	16#F85A: F_AX5xErrMsg:= 'F85A =  One cable feedback: Parameter data access error - Timeout';
	16#F85B: F_AX5xErrMsg:= 'F85B =  One cable feedback: Parameter data access error';
	16#F85C: F_AX5xErrMsg:= 'F85C =  One cable feedback: Internal error';
	16#F85D: F_AX5xErrMsg:= 'F85D =  One cable feedback: Encoder status signals an error';
	16#F85E: F_AX5xErrMsg:= 'F85E =  OCT / HpfDSL: Long message bad answer';
	16#F85F: F_AX5xErrMsg:= 'F85F =  OCT / HpfDSL: Shutdown of the encoder failed';
	16#F860: F_AX5xErrMsg:= 'F860 =  OCT / HpfDSL: File write failed.';
	16#F861: F_AX5xErrMsg:= 'F861 =  OCT / HpfDSL: Invalid serial number.';
	16#F862: F_AX5xErrMsg:= 'F862 =  OCT / HpfDSL: No access to the motor temperature sensor.';
	16#F863: F_AX5xErrMsg:= 'F863 =  OCT / HpfDSL: Invalid edge register value.';
	16#F864: F_AX5xErrMsg:= 'F864 =  OCT / HpfDSL: Read cyclic data, Request error';
	16#F865: F_AX5xErrMsg:= 'F865 =  OCT / HpfDSL: Feedback not found.';
	16#F866: F_AX5xErrMsg:= 'F866 =  OCT / HpfDSL: No electronic data sheet found.';
	16#F867: F_AX5xErrMsg:= 'F867 =  OCT / HpfDSL: The electronic data sheet is invalid.';
	16#F868: F_AX5xErrMsg:= 'F868 =  OCT / HpfDSL: User data file invalid.';
	16#F869: F_AX5xErrMsg:= 'F869 =  OCT / HpfDSL: Position offset file invalid.';
	16#F86A: F_AX5xErrMsg:= 'F86A =  OCT / HpfDSL: Commutation offset file invalid.';
	16#F86B: F_AX5xErrMsg:= 'F86B =  OCT / HpfDSL: Invalid file header.';
	16#F86C: F_AX5xErrMsg:= 'F86C =  OCT / HpfDSL: Invalid file.';
	16#F86D: F_AX5xErrMsg:= 'F86D =  OCT / HpfDSL: Position deviation monitoring: Value too many cycles not zero.';
	16#F86E: F_AX5xErrMsg:= 'F86E =  OCT / HpfDSL: Detailed error info';
	16#F86F: F_AX5xErrMsg:= 'F86F =  OCT / HpfDSL: Initial encoder status error';
	16#F870: F_AX5xErrMsg:= 'F870 =  Feedback "AX572x": Encoder not ready';
	16#F872: F_AX5xErrMsg:= 'F872 =  Feedback "AX572x": Position is invalid';
	16#F873: F_AX5xErrMsg:= 'F873 =  Feedback "AX572x": Position is invalid';
	16#F874: F_AX5xErrMsg:= 'F874 =  Feedback "AX572x": Feedbackregister invalid';
	16#F875: F_AX5xErrMsg:= 'F875 =  Feedback "AX572x": Unexpected encoder';
	16#F876: F_AX5xErrMsg:= 'F876 =  Feedback "EnDat 2.2": UART-error';
	16#F877: F_AX5xErrMsg:= 'F877 =  Feedback "AX572x": Out of memory';
	16#F879: F_AX5xErrMsg:= 'F879 =  Feedback "AX572x": Supply voltage';
	16#F87A: F_AX5xErrMsg:= 'F87A =  Feedback "AX572x": Defective Powerup Phase of the feedback system';
	16#F87C: F_AX5xErrMsg:= 'F87C =  Feedback "AX572x": FB protocol not supported';
	16#F87D: F_AX5xErrMsg:= 'F87D =  Feedback "AX572x": Parameter error';
	16#F880: F_AX5xErrMsg:= 'F880 =  HTL: Encoder not ready.';
	16#F881: F_AX5xErrMsg:= 'F881 =  HTL: Error flag active.';
	16#F882: F_AX5xErrMsg:= 'F882 =  HTL: Wrong interface.';
	16#F883: F_AX5xErrMsg:= 'F883 =  HTL: Timeout.';
	16#F8A0: F_AX5xErrMsg:= 'F8A0 =  OCT / HpfDSL: Default state entered.';
	16#F8A1: F_AX5xErrMsg:= 'F8A1 =  OCT / HpfDSL: sHub not supported.';
	16#FA00: F_AX5xErrMsg:= 'FA00 =  Feedback process channel error.';
	16#FA01: F_AX5xErrMsg:= 'FA01 =  Feedback process data channel init error';
	16#FA02: F_AX5xErrMsg:= 'FA02 =  Feedback process channel init command timeout.';
	16#FA03: F_AX5xErrMsg:= 'FA03 =  Feedback process channel init command not idle.';
	16#FA04: F_AX5xErrMsg:= 'FA04 =  Feedback process channel init error.';
	16#FA05: F_AX5xErrMsg:= 'FA05 =  Feedback process channel init error.';
	16#FA06: F_AX5xErrMsg:= 'FA06 =  Feedback process channel init error.';
	16#FA07: F_AX5xErrMsg:= 'FA07 =  Feedback process channel,  unknown feedback type.';
	16#FA40: F_AX5xErrMsg:= 'FA40 =  Feedback process channel error (1Vss)';
	16#FA41: F_AX5xErrMsg:= 'FA41 =  Feedback process channel error (1Vss)';
	16#FA42: F_AX5xErrMsg:= 'FA42 =  Feedback process channel error (1Vss)';
	16#FA43: F_AX5xErrMsg:= 'FA43 =  Feedback process channel error (1Vss)';
	16#FA44: F_AX5xErrMsg:= 'FA44 =  Feedback process channel error (1Vss)';
	16#FA45: F_AX5xErrMsg:= 'FA45 =  Feedback process channel error (1Vss)';
	16#FA46: F_AX5xErrMsg:= 'FA46 =  Feedback process channel error (1Vss)';
	16#FA47: F_AX5xErrMsg:= 'FA47 =  Feedback process channel error (1Vss)';
	16#FA48: F_AX5xErrMsg:= 'FA48 =  Feedback process channel error (1Vss)';
	16#FA49: F_AX5xErrMsg:= 'FA49 =  Feedback process channel error (1Vss)';
	16#FA4A: F_AX5xErrMsg:= 'FA4A =  Feedback process channel error (1Vss)';
	16#FA4B: F_AX5xErrMsg:= 'FA4B =  Feedback process channel error (1Vss)';
	16#FA4C: F_AX5xErrMsg:= 'FA4C =  Feedback process channel error. Failed to set the reference voltage.';
	16#FA4D: F_AX5xErrMsg:= 'FA4D =  Feedback process channel error. Firmware index not valid.';
	16#FA60: F_AX5xErrMsg:= 'FA60 =  Feedback error TTL: System error';
	16#FA61: F_AX5xErrMsg:= 'FA61 =  Feedback error TTL: Unknown state';
	16#FA62: F_AX5xErrMsg:= 'FA62 =  Feedback error TTL: Qudarature encoder error';
	16#FA63: F_AX5xErrMsg:= 'FA63 =  Feedback error TTL: Quadrant init error';
	16#FA64: F_AX5xErrMsg:= 'FA64 =  Feedback error TTL: Reference voltage error';
	16#FA65: F_AX5xErrMsg:= 'FA65 =  Feedback error TTL: Firmware index not supported';
	16#FA80: F_AX5xErrMsg:= 'FA80 =  Feedback "Resolver": Got no timer';
	16#FA81: F_AX5xErrMsg:= 'FA81 =  Feedback "Resolver": Unknown state';
	16#FA82: F_AX5xErrMsg:= 'FA82 =  Feedback "Resolver": Initialisation of the sampling instance failed';
	16#FA83: F_AX5xErrMsg:= 'FA83 =  Feedback "Resolver": Calibration incorrect';
	16#FA84: F_AX5xErrMsg:= 'FA84 =  Feedback "Resolver": Number of poles not supported.';
	16#FA85: F_AX5xErrMsg:= 'FA85 =  Feedback "Resolver": Excitation frequence not supported';
	16#FA86: F_AX5xErrMsg:= 'FA86 =  Feedback "Resolver": Transformation ratio not supported.';
	16#FA87: F_AX5xErrMsg:= 'FA87 =  Feedback "Resolver": Connector not supported.';
	16#FA88: F_AX5xErrMsg:= 'FA88 =  Feedback "Resolver": Invalid ADC configuration';
	16#FA89: F_AX5xErrMsg:= 'FA89 =  Feedback "Resolver": ADC time out';
	16#FA8A: F_AX5xErrMsg:= 'FA8A =  Feedback "Resolver": Hardware does not support a resolver';
	16#FA8B: F_AX5xErrMsg:= 'FA8B =  Feedback "Resolver": Amplitude of the resolver output voltage too large';
	16#FA8C: F_AX5xErrMsg:= 'FA8C =  Feedback "Resolver": Amplitude of the resolver output voltage too low';
	16#FA8D: F_AX5xErrMsg:= 'FA8D =  Feedback "Resolver": Hardware does not support a resolver';
	16#FA8E: F_AX5xErrMsg:= 'FA8E =  Feedback "Resolver": Internal error';
	16#FA8F: F_AX5xErrMsg:= 'FA8F =  Feedback "Resolver": Feedback gear not supported.';
	16#FA90: F_AX5xErrMsg:= 'FA90 =  Feedback "Resolver": Amplitude correction limit exceeded.';
	16#FA91: F_AX5xErrMsg:= 'FA91 =  Feedback "Resolver": Use of reserved parameter.';
	16#FA92: F_AX5xErrMsg:= 'FA92 =  Feedback "Resolver": Offset out of range.';
	16#FA93: F_AX5xErrMsg:= 'FA93 =  Feedback "Resolver": Offset balance failed';
	16#FA94: F_AX5xErrMsg:= 'FA94 =  Feedback "Resolver": Invalid cycle time configuration.';
	16#FA95: F_AX5xErrMsg:= 'FA95 =  Feedback "Resolver": Internal Error';
	16#FA96: F_AX5xErrMsg:= 'FA96 =  Feedback "Resolver": Phase Calibration - Amplitude too low';
	16#FA97: F_AX5xErrMsg:= 'FA97 =  Feedback "Resolver": Phase Calibration - Amplitude too high';
	16#FAB0: F_AX5xErrMsg:= 'FAB0 =  Feedback "MES": Unknown state';
	16#FAB1: F_AX5xErrMsg:= 'FAB1 =  Feedback "MES": Connector not supported.';
	16#FAB2: F_AX5xErrMsg:= 'FAB2 =  Feedback "MES": Invalid ADC configuration';
	16#FAB3: F_AX5xErrMsg:= 'FAB3 =  Feedback "MES": ADC time out';
	16#FAB4: F_AX5xErrMsg:= 'FAB4 =  Feedback "MES": Hardware does not support a MES';
	16#FAB5: F_AX5xErrMsg:= 'FAB5 =  Feedback "MES": Output voltage too high';
	16#FAB6: F_AX5xErrMsg:= 'FAB6 =  Feedback "MES": Output voltage too low';
	16#FAB7: F_AX5xErrMsg:= 'FAB7 =  Feedback "MES": Hardware does not support a MES';
	16#FAB8: F_AX5xErrMsg:= 'FAB8 =  Feedback "MES": Internal error';
	16#FAB9: F_AX5xErrMsg:= 'FAB9 =  Feedback "MES": Feedback gear not supported.';
	16#FABA: F_AX5xErrMsg:= 'FABA =  Feedback "MES": Amplitude correction limit exceeded.';
	16#FABB: F_AX5xErrMsg:= 'FABB =  Feedback "MES": Use of reserved parameter.';
	16#FABC: F_AX5xErrMsg:= 'FABC =  Feedback "MES": Invalid cycle time configuration.';
	16#FC00: F_AX5xErrMsg:= 'FC00 =  Fpga error';
	16#FC01: F_AX5xErrMsg:= 'FC01 =  Fpga error';
	16#FC02: F_AX5xErrMsg:= 'FC02 =  Fpga error';
	16#FC03: F_AX5xErrMsg:= 'FC03 =  Control voltage error: undervoltage';
	16#FC04: F_AX5xErrMsg:= 'FC04 =  Driver unit error: undervoltage';
	16#FC05: F_AX5xErrMsg:= 'FC05 =  Dsp watchdog error.';
	16#FC06: F_AX5xErrMsg:= 'FC06 =  Dsp clock error.';
	16#FC07: F_AX5xErrMsg:= 'FC07 =  ESC clock error.';
	16#FC08: F_AX5xErrMsg:= 'FC08 =  Overcurrent error';
	16#FC09: F_AX5xErrMsg:= 'FC09 =  Deadtime error.';
	16#FC0A: F_AX5xErrMsg:= 'FC0A =  Lock error.';
	16#FC0B: F_AX5xErrMsg:= 'FC0B =  Overcurrent error motor,  short curcuit detection (X13 / X23).';
	16#FC0C: F_AX5xErrMsg:= 'FC0C =  Safety card activated';
	16#FC0D: F_AX5xErrMsg:= 'FC0D =  Shorted coils brake triggerd by the FPGA logic.';
	16#FC0E: F_AX5xErrMsg:= 'FC0E =  Torque off triggerd by the FPGA logic.';
	16#FC0F: F_AX5xErrMsg:= 'FC0F =  FPGA logic: Brake chopper error';
	16#FC10: F_AX5xErrMsg:= 'FC10 =  FPGA logic: Motorcurrent sum error.';
	16#FC11: F_AX5xErrMsg:= 'FC11 =  FPGA logic: Powersupply error.';
	16#FC12: F_AX5xErrMsg:= 'FC12 =  FPGA logic: Umains phase error.';
	16#FC13: F_AX5xErrMsg:= 'FC13 =  FPGA logic:DC link overvoltage';
	16#FC30: F_AX5xErrMsg:= 'FC30 =  Internal error (I2C)';
	16#FC31: F_AX5xErrMsg:= 'FC31 =  Internal error (I2C)';
	16#FC32: F_AX5xErrMsg:= 'FC32 =  Internal error (I2C)';
	16#FC33: F_AX5xErrMsg:= 'FC33 =  Internal error (I2C)';
	16#FC34: F_AX5xErrMsg:= 'FC34 =  Internal error (I2C)';
	16#FC35: F_AX5xErrMsg:= 'FC35 =  Internal error (I2C)';
	16#FC36: F_AX5xErrMsg:= 'FC36 =  Internal error (I2C)';
	16#FC37: F_AX5xErrMsg:= 'FC37 =  Internal communication error';
	16#FC38: F_AX5xErrMsg:= 'FC38 =  Error reading error stack.';
	16#FC39: F_AX5xErrMsg:= 'FC39 =  Error reading operation time.';
	16#FC3A: F_AX5xErrMsg:= 'FC3A =  Error reading eeprom.';
	16#FC3B: F_AX5xErrMsg:= 'FC3B =  Error reading error stack.';
	16#FC3C: F_AX5xErrMsg:= 'FC3C =  Error reading error stack.';
	16#FC3D: F_AX5xErrMsg:= 'FC3D =  Error reading operation time.';
	16#FC3E: F_AX5xErrMsg:= 'FC3E =  Error reading factory settings.';
	16#FC3F: F_AX5xErrMsg:= 'FC3F =  Error reading factory settings.';
	16#FC40: F_AX5xErrMsg:= 'FC40 =  Error saving Hw-Id.';
	16#FC41: F_AX5xErrMsg:= 'FC41 =  Error saving Hw-Id.';
	16#FC42: F_AX5xErrMsg:= 'FC42 =  Error saving factory settings.';
	16#FC43: F_AX5xErrMsg:= 'FC43 =  Error saving factory settings.';
	16#FC44: F_AX5xErrMsg:= 'FC44 =  Error clearing operation time.';
	16#FC45: F_AX5xErrMsg:= 'FC45 =  Error clearing error list.';
	16#FC46: F_AX5xErrMsg:= 'FC46 =  Error reading operation time.';
	16#FC47: F_AX5xErrMsg:= 'FC47 =  Error clearing error stack.';
	16#FC70: F_AX5xErrMsg:= 'FC70 =  Init of the keypad failed.';
	16#FC80: F_AX5xErrMsg:= 'FC80 =  Probe unit error.';
	16#FC81: F_AX5xErrMsg:= 'FC81 =  Probe unit error.';
	16#FC82: F_AX5xErrMsg:= 'FC82 =  Probe unit error.';
	16#FC83: F_AX5xErrMsg:= 'FC83 =  Invalid probe unit configuration';
	16#FC84: F_AX5xErrMsg:= 'FC84 =  Probe unit configuration: Activate signal configuration error.';
	16#FCB0: F_AX5xErrMsg:= 'FCB0 =  LCD Display init failed.';
	16#FCB1: F_AX5xErrMsg:= 'FCB1 =  LDC Display error.';
	16#FCB2: F_AX5xErrMsg:= 'FCB2 =  LDC Display error.';
	16#FCB3: F_AX5xErrMsg:= 'FCB3 =  LCD-Display: Initialisierungsfehler';
	16#FCB4: F_AX5xErrMsg:= 'FCB4 =  LCD-Display: Time out';
	16#FCD0: F_AX5xErrMsg:= 'FCD0 =  Positive limit switch error.';
	16#FCD1: F_AX5xErrMsg:= 'FCD1 =  Negative limit switch error.';
	16#FCD2: F_AX5xErrMsg:= 'FCD2 =  Overspeed error.';
	16#FCD3: F_AX5xErrMsg:= 'FCD3 =  Overspeed error.';
	16#FCD4: F_AX5xErrMsg:= 'FCD4 =  AX5000 utilization error.';
	16#FCD5: F_AX5xErrMsg:= 'FCD5 =  Current limitation: U/F error';
	16#FCD6: F_AX5xErrMsg:= 'FCD6 =  Monitoring functions: Shorted coil / DC brake error';
	16#FCD7: F_AX5xErrMsg:= 'FCD7 =  Maximum output frequency limit exceeded.';
	16#FD00: F_AX5xErrMsg:= 'FD00 =  Motor management: Init failed';
	16#FD01: F_AX5xErrMsg:= 'FD01 =  Motor management: Init failed';
	16#FD03: F_AX5xErrMsg:= 'FD03 =  Brake management error.';
	16#FD04: F_AX5xErrMsg:= 'FD04 =  Periphery voltage missing.';
	16#FD05: F_AX5xErrMsg:= 'FD05 =  Motor management error.';
	16#FD06: F_AX5xErrMsg:= 'FD06 =  Motor management error.';
	16#FD07: F_AX5xErrMsg:= 'FD07 =  Motor overtemperature shut down.';
	16#FD08: F_AX5xErrMsg:= 'FD08 =  Motor management: Drive type don"t match.';
	16#FD09: F_AX5xErrMsg:= 'FD09 =  Motor management: Motor type don"t match.';
	16#FD0A: F_AX5xErrMsg:= 'FD0A =  Configured channel peak current is greater than the motor peak current.';
	16#FD0B: F_AX5xErrMsg:= 'FD0B =  Configured channel peak current is greater than the amplifier channel peak current.';
	16#FD0C: F_AX5xErrMsg:= 'FD0C =  Configured channel current is greater than the motor coninuous stall current.';
	16#FD0D: F_AX5xErrMsg:= 'FD0D =  Configured channel current is greater than the amplifier rated current.';
	16#FD0E: F_AX5xErrMsg:= 'FD0E =  Invalid total output current.';
	16#FD0F: F_AX5xErrMsg:= 'FD0F =  Motor brake: Current monitoring error.';
	16#FD10: F_AX5xErrMsg:= 'FD10 =  Periphery voltage too high.';
	16#FD11: F_AX5xErrMsg:= 'FD11 =  Periphery voltage too low.';
	16#FD12: F_AX5xErrMsg:= 'FD12 =  Unknown constraint IDN';
	16#FD13: F_AX5xErrMsg:= 'FD13 =  Too low dielectric strength of the motor winding.';
	16#FD14: F_AX5xErrMsg:= 'FD14 =  Constraint check failed.';
	16#FD15: F_AX5xErrMsg:= 'FD15 =  The maximum feedback frequency is too high.';
	16#FD16: F_AX5xErrMsg:= 'FD16 =  Unknown feedback system.';
	16#FD17: F_AX5xErrMsg:= 'FD17 =  Motor overload shutdown.';
	16#FD18: F_AX5xErrMsg:= 'FD18 =  Motorbrake current: Measuring error';
	16#FD19: F_AX5xErrMsg:= 'FD19 =  A/D-Converter: Peripheral voltage - measuring error';
	16#FD1A: F_AX5xErrMsg:= 'FD1A =  A/D-Converter: Motor temperature - measuring error';
	16#FD1B: F_AX5xErrMsg:= 'FD1B =  Motor cont. stall torque > peak torque';
	16#FD1C: F_AX5xErrMsg:= 'FD1C =  ASM don"t support"s usage of P-0-0077';
	16#FD1D: F_AX5xErrMsg:= 'FD1D =  Invalid torque characteristic data.';
	16#FD1E: F_AX5xErrMsg:= 'FD1E =  Invalid inductance characteristic data.';
	16#FD1F: F_AX5xErrMsg:= 'FD1F =  Got no memory.';
	16#FD20: F_AX5xErrMsg:= 'FD20 =  Motor management: Invalid motor data.';
	16#FD21: F_AX5xErrMsg:= 'FD21 =  Motor management: Voltage error';
	16#FD22: F_AX5xErrMsg:= 'FD22 =  Motor management: Current error';
	16#FD40: F_AX5xErrMsg:= 'FD40 =  Power management: Init failed';
	16#FD41: F_AX5xErrMsg:= 'FD41 =  Mains supply: U mains too high.';
	16#FD42: F_AX5xErrMsg:= 'FD42 =  Mains supply: U mains too low.';
	16#FD43: F_AX5xErrMsg:= 'FD43 =  Mains supply: Power down.';
	16#FD44: F_AX5xErrMsg:= 'FD44 =  Mains supply: Phase error.';
	16#FD45: F_AX5xErrMsg:= 'FD45 =  Continous power internal brake resistor too low.';
	16#FD46: F_AX5xErrMsg:= 'FD46 =  Power management error.';
	16#FD47: F_AX5xErrMsg:= 'FD47 =  Power management error.';
	16#FD48: F_AX5xErrMsg:= 'FD48 =  Power management error.';
	16#FD49: F_AX5xErrMsg:= 'FD49 =  IGBT temperature measuring error.';
	16#FD4A: F_AX5xErrMsg:= 'FD4A =  IGBT temperature measuring error.';
	16#FD4B: F_AX5xErrMsg:= 'FD4B =  DC link undervoltage.';
	16#FD4C: F_AX5xErrMsg:= 'FD4C =  DC link overvoltage';
	16#FD4D: F_AX5xErrMsg:= 'FD4D =  Cooling error shut down.';
	16#FD4E: F_AX5xErrMsg:= 'FD4E =  Control voltage error';
	16#FD4F: F_AX5xErrMsg:= 'FD4F =  Overvoltage error.';
	16#FD50: F_AX5xErrMsg:= 'FD50 =  Undervoltage error.';
	16#FD51: F_AX5xErrMsg:= 'FD51 =  Power supply phase error.';
	16#FD52: F_AX5xErrMsg:= 'FD52 =  Unknown internal brake resistor.';
	16#FD53: F_AX5xErrMsg:= 'FD53 =  U_mains power up after mains power failure.';
	16#FD54: F_AX5xErrMsg:= 'FD54 =  Unknown nominal device current.';
	16#FD55: F_AX5xErrMsg:= 'FD55 =  AX5021: Brake resistor overtemperature shut down';
	16#FD56: F_AX5xErrMsg:= 'FD56 =  Error Power Management: Transfer error, unknown channel.';
	16#FD57: F_AX5xErrMsg:= 'FD57 =  Error Power Management: Load resistor active and axis enabled';
	16#FD58: F_AX5xErrMsg:= 'FD58 =  Error Power Management: Check external dc link connection';
	16#FD59: F_AX5xErrMsg:= 'FD59 =  Error Power Management: Wrong external brake resistor found';
	16#FD5A: F_AX5xErrMsg:= 'FD5A =  Power Management: Overcurrent - dc link connection';
	16#FD80: F_AX5xErrMsg:= 'FD80 =  System time underflow error.';
	16#FD81: F_AX5xErrMsg:= 'FD81 =  Wrong timer pointer.';
	16#FD82: F_AX5xErrMsg:= 'FD82 =  Out of timer.';
	16#FD83: F_AX5xErrMsg:= 'FD83 =  Invalid identity object type.';
	16#FD84: F_AX5xErrMsg:= 'FD84 =  Invalid firmware index.';
	16#FD85: F_AX5xErrMsg:= 'FD85 =  Feedback firmware checksum error.';
	16#FD86: F_AX5xErrMsg:= 'FD86 =  System timer underflow.';
	16#FD87: F_AX5xErrMsg:= 'FD87 =  Error: Out of system timer.';
	16#FD88: F_AX5xErrMsg:= 'FD88 =  Found not supported hardware type.';
	16#FD89: F_AX5xErrMsg:= 'FD89 =  Safety card type not supported.';
	16#FD8A: F_AX5xErrMsg:= 'FD8A =  Option card: Type not supported';
	16#FD8B: F_AX5xErrMsg:= 'FD8B =  Option card: Interface Id is not supported.';
	16#FD8C: F_AX5xErrMsg:= 'FD8C =  Option card: Channel count is not supported.';
	16#FD8D: F_AX5xErrMsg:= 'FD8D =  Invalid identity object';
	16#FD8E: F_AX5xErrMsg:= 'FD8E =  Optioncard: Interface of the FPGA 2 not supported';
	16#FDB0: F_AX5xErrMsg:= 'FDB0 =  Customer specific function: Init failed.';
	16#FDC0: F_AX5xErrMsg:= 'FDC0 =  Internal command state machine error.';
	16#FDC1: F_AX5xErrMsg:= 'FDC1 =  Internal command state machine error.';
	16#FDC2: F_AX5xErrMsg:= 'FDC2 =  Internal command state machine error.';
	16#FDC3: F_AX5xErrMsg:= 'FDC3 =  Internal command state machine error.';
	16#FDD0: F_AX5xErrMsg:= 'FDD0 =  Safety card: Unknown hardware type.';
	16#FDD1: F_AX5xErrMsg:= 'FDD1 =  Safety: internal error, out of memory';
	16#FDD2: F_AX5xErrMsg:= 'FDD2 =  Safety: internal error, got no timer';
	16#FDD3: F_AX5xErrMsg:= 'FDD3 =  Safety switch off while the axis was enabled.';
	16#FDD4: F_AX5xErrMsg:= 'FDD4 =  Configured safety option don"t match';
	16#FDD5: F_AX5xErrMsg:= 'FDD5 =  The basic unit of the drive dont supports a safety option.';
	16#FDD6: F_AX5xErrMsg:= 'FDD6 =  Safety Option: Not supported firmware index.';
	16#FDD7: F_AX5xErrMsg:= 'FDD7 =  Safety slot: No safety or dummy card inserted';
	16#FDD8: F_AX5xErrMsg:= 'FDD8 =  Safety slot: Wrong safety or dummy card inserted';
	16#FDD9: F_AX5xErrMsg:= 'FDD9 =  Safety card: safety card activated - internal reaction';
	16#FDDA: F_AX5xErrMsg:= 'FDDA =  Safety slot: Wrong safety card AX5805 or AX5806 inserted';
	16#FDDB: F_AX5xErrMsg:= 'FDDB =  Safety card: Internal error.';
	16#FFFE: F_AX5xErrMsg:= 'FFFE =  Missing implementation!';
	
ELSE
	F_AX5xErrMsg := UINT_TO_STRING(uiDriveError);
	F_AX5xErrMsg := concat(F_AX5xErrMsg, ' Unknown Error code');
END_CASE
F_AX5xErrMsg := F_AX5xErrMsg;

END_FUNCTION

// ---- POUs/P_ModeStateManager.TcPOU
//==================================================================================================
//							Beckhoff Automation Poland
//									2.11.2018
//	Zarzadzeni trybami pracy i komendami - Satate Machine
// 	v1.2	|| TC v 3.1.4022.25		|| - dodano Initialization 
// 	v1.1	|| TC v 3.1.4022.4		|| - Aktualizacja - dodano test Abort z HMI 
// 	v1.0	|| TC v 3.1.4022.4		|| - Pierwsza wersja
//==================================================================================================
PROGRAM P_ModeStateManager
VAR
	//	GVL_Machine - HMI handling
	bHMIModeRequest_Automatic			: BOOL;
	bHMIModeRequest_Manual				: BOOL;
	bHMIModeRequest_Maintenance			: BOOL;
	
	bHMICommandRequest_Run				: BOOL;
	bHMICommandRequest_Stop				: BOOL;
	bHMICommandRequest_Reset			: BOOL;
	bHMICommandRequest_Restart			: BOOL;
	bHMICommandRequest_Abort			: BOOL;
	// Rising edge detection
	rtButtonAutomatic					: R_TRIG;
	rtButtonManual						: R_TRIG;
	rtButtonMaintenance					: R_TRIG;
	rtButtonStart						: R_TRIG;
	rtButtonReset						: R_TRIG;
	rtButtonStop						: R_TRIG;
	// State change permissions
	bAllowChangeToManual				: BOOL;
	bAllowChangeToMaintenance			: BOOL;
	bAllowChangeToAutomatic				: BOOL;
END_VAR

// Triggers
rtButtonAutomatic(CLK:= bHMIModeRequest_Automatic);
rtButtonManual(CLK:= bHMIModeRequest_Manual);
rtButtonMaintenance(CLK:= bHMIModeRequest_Maintenance);
rtButtonStart(CLK:= GVL_IO.di_PBStart OR bHMICommandRequest_Run);
rtButtonStop(CLK:= GVL_IO.di_PBStop OR bHMICommandRequest_Stop);
rtButtonReset(CLK:= GVL_IO.di_PBReset OR bHMICommandRequest_Reset);

// SAFETY niezaleznie
IF NOT GVL_IO.bSAFETY_PermissionSS1 OR bHMICommandRequest_Abort THEN
	GVL_Machine.eCommand						:= E_MachineCommand.eAbort;
	GVL_Machine.eState							:= E_MachineState.eAborted;
END_IF
		
CASE GVL_Machine.eMode OF 

	E_MachineMode.eInitialization:

		// Reset just in case of init error
		P_Initialization(bReset := (P_Initialization.bError AND rtButtonReset.Q), bTestMode := );
		IF P_Initialization.bInitialized THEN
			// Choose mode to go
			GVL_Machine.eMode						:= E_MachineMode.eManual;
		END_IF
		
	E_MachineMode.eAutomatic:

		// Zmiana trybu tylko gdy maszyna nie jest w Running
		IF GVL_Machine.eState <> E_MachineState.eRunning THEN
			IF rtButtonMaintenance.Q THEN
				GVL_Machine.eState				:= E_MachineState.eIdle;
				GVL_Machine.eMode				:= E_MachineMode.eMaintenance;
			END_IF
		END_IF

		//==============================================
		IF rtButtonStart.Q THEN 
			GVL_Machine.eCommand 	:= E_MachineCommand.eRun;
		END_IF

		IF rtButtonReset.Q AND GVL.bRestartRequired THEN
			GVL_Machine.eCommand	:= E_MachineCommand.eRestart;
		END_IF
		
		IF rtButtonReset.Q AND NOT GVL.bRestartRequired THEN
			GVL_Machine.eCommand	:= E_MachineCommand.eReset;
		END_IF
		
		IF GVL.bGeneralError OR GVL.bGeneralFatalError OR rtButtonStop.Q THEN
			GVL_Machine.eCommand	:= E_MachineCommand.eStop ;
		END_IF
		
	E_MachineMode.eMaintenance, E_MachineMode.eManual:
	
		// Reset, Restart, Error - not used
		
		// Zmiana trybu tylko gdy maszyna nie jest w Running
		IF GVL_Machine.eState <> E_MachineState.eRunning THEN
			IF rtButtonAutomatic.Q (* OR sth *) THEN
				GVL_Machine.eState				:= E_MachineState.eIdle;
				GVL_Machine.eMode				:= E_MachineMode.eAutomatic;
			END_IF
		END_IF
		
		//==============================================
		IF rtButtonStart.Q THEN 
			GVL_Machine.eCommand 	:= E_MachineCommand.eRun;
		END_IF

		IF rtButtonReset.Q AND GVL.bRestartRequired THEN
			GVL_Machine.eCommand	:= E_MachineCommand.eRestart;
		END_IF
		
		IF rtButtonReset.Q AND NOT GVL.bRestartRequired THEN
			GVL_Machine.eCommand	:= E_MachineCommand.eReset;
		END_IF
		
		IF rtButtonStop.Q THEN
			GVL_Machine.eCommand	:= E_MachineCommand.eStop ;
		END_IF

END_CASE

ACTION Act_CollectMachineState:
// Action to decide global machine state
GVL_Machine.eState; // :=
END_ACTION

ACTION Act_ModeChangeSelector:
bAllowChangeToManual 				:= NOT (P_Template.eMachineState <> E_MachineState.eRunning); //
bAllowChangeToMaintenance;
bAllowChangeToAutomatic;
END_ACTION

END_PROGRAM

// ---- POUs/P_Initialization.TcPOU
//==================================================================================================
//							Beckhoff Automation Poland
//									2.11.2018
//	Program inicjalizujacy prace maszyny - powinien byc wykonywany tylko w trybie E_MachineMode.eInitialization
//	Przejscie do innych trybow powinno byc mozliwe po wystawieniu flagi bInitialized
//	Program podczas inicjalizacji tlumi globalne flagi: GVL.bMuteGeneralError i GVL.bMuteGeneralFatalError
//	Reset mozliwy tylko w przypadku bledu.
//	Zawiera opsje testu - ignorujemy wowczas bledy i przechodzimy od razu do stanu bInitialized
// 	v1.0	|| TC v 3.1.4022.25		|| - Pierwsza wersja
//==================================================================================================
PROGRAM P_Initialization
VAR_INPUT
	bReset					: BOOL;
	bTestMode				: BOOL;				// Deactivate error detecton - go to initialized
END_VAR
VAR_OUTPUT
	bInitialized			: BOOL;
	bBusy					: BOOL;
	bError					: BOOL;
END_VAR
VAR
	iStep					: INT;
	rtReset					: R_TRIG;
	rtError					: R_TRIG;
	tonWatchdog				: TON;
END_VAR

// Wait some time to initialize
tonWatchdog(IN:= bBusy, PT:= T#1M, Q=> , ET=> );
rtError(CLK:= tonWatchdog.Q, Q=> );

IF rtError.Q THEN
	iStep							:= 1000;
END_IF

// Reset - reinitialize
rtReset(CLK:= bReset, Q=> );

IF bTestMode THEN
	iStep							:= 500;
END_IF

CASE iStep OF

	0: // Idle
	
		iStep	 					:= iStep + 10;
	
	10: 
	
		IF P_SystemInfo.bOK THEN
			iStep 					:= iStep + 10;
		ELSE
			// There is problem with System - usually persistent data
			P_SystemInfo.bConfirm 	:= bReset;
		END_IF
	
	20:

		IF P_EtherCAT_Diag.bOK THEN
			iStep 					:= iStep + 10;
		END_IF

	30:

		IF P_Checks.bOK THEN
			iStep 					:= iStep + 10;
		END_IF
		
	40:

		IF P_TaskInfo.bOK THEN
			iStep 					:= iStep + 10;
		END_IF
		
	50:
	// Serial No, etc
		iStep 						:= 500;
		
	500: // Initialized
	
		;
	
	1000: // Error step, wait for reset
	
		IF rtReset.Q THEN
			P_SystemInfo.bConfirm 	:= TRUE;
			iStep 					:= 0;
		END_IF;

END_CASE

bBusy 								:= iStep < 500;
bError 								:= iStep = 1000;
bInitialized						:= iStep = 500;

// Mute Errors during init phase
GVL.bMuteGeneralError				:= bBusy;
GVL.bMuteGeneralFatalError			:= bBusy;

END_PROGRAM

// ---- POUs/POUsAxisOnline/AX8000/FB_HoldingBrakeCtrlAX8000.TcPOU
//==================================================================================================
//							Beckhoff Automation Poland
//									12.04.2018
//	Blok funkcyjny kontroli luzownika w silniku podpietym do AX8000. Przewaga ForceLock
//	Dzialania na obiekcie: 3000:07 Motor brake force
//	Index:			AxisMainSlot: 16#3000 (Ch A)/ 16#3400 (Ch B)
//	Subindex:		16#07
//	Datatype:		ENUM (INT16)
//	Enum Value:		0 (0x00): 	Release_force
//					1 (0x01): 	Force_lock
//					2 (0x02): 	Force_unlock
//
//  v1.0	|| TC v 3.1.4022.16		|| - pierwsza wersja
//==================================================================================================
FUNCTION_BLOCK FB_HoldingBrakeCtrlAX8000
VAR_INPUT
	bForceLock 						: BOOL;								// 
	bForceUnlock					: BOOL;								// 
	stDriveRef						: ST_DriveRef;
END_VAR
VAR_OUTPUT
	bBusy							: BOOL;
	bError							: BOOL; 							// General error: parameter or CoE read.
																		// If bError = TRUE and bInitialized = FALSE - error during read motor data.
																		// If bError = TRUE and bInitialized = TRUE and (iAdsErrId <> 0 or iCANopenErrId <> 0) then I2T read error
																		// If bError = TRUE and bInitialized = TRUE and iAdsErrId = 0 and iCANopenErrId = 0 then parameter error: rTorqueLimit outside permitted range rTorqueLimitLow..rTorqueLimitHigh or Empty stDriveRef
	iAdsErrId						: UINT;								// Forwarded output FB_CoERead_ByDriveRef
	iCANopenErrId					: UINT;								// Forwarded output FB_CoERead_ByDriveRef
END_VAR
VAR
	bExecute						: BOOL;
	iMotorBrakeForce				: INT;								// 0 - Release_force, 1 - Force_lock, 2 - Force_unlock
	rtForceLock						: R_TRIG;
	rtForceUnlock					: R_TRIG;
	ftForceLock						: F_TRIG;
	ftForceUnlock					: F_TRIG;
	fbForceLockUnlock				: FB_CoEWrite_ByDriveRef;
END_VAR

{region "Call triggers"}
//======================= Call triggers =========================
rtForceLock(CLK:= bForceLock);
ftForceLock(CLK:= bForceLock);
rtForceUnlock(CLK:= bForceUnlock);
ftForceUnlock(CLK:= bForceUnlock);
bExecute								:= rtForceLock.Q OR ftForceLock.Q OR rtForceUnlock.Q OR ftForceUnlock.Q;
//===============================================================
{endregion}
{region "Main code"}
//========================= Main code ===========================
IF bExecute THEN
	iMotorBrakeForce 						:= 0;										// Clear value
	iMotorBrakeForce.1 						:= bForceUnlock;							// Set force unlock bit
	iMotorBrakeForce 						:= SEL(bForceLock, iMotorBrakeForce, 1);	// Set force lock bit, it has higher priority than unlock
END_IF

fbForceLockUnlock(	stDriveRef				:= stDriveRef, 
					nIndex					:= 16#3000 + (stDriveRef.nDriveNo * 16#400), 
					nSubIndex				:= 16#07, 
					pSrcBuf					:= ADR(iMotorBrakeForce), 
					cbBufLen				:= SIZEOF(iMotorBrakeForce), 
					bExecute				:= bExecute,
					bBusy					=> bBusy, 
					bError					=> bError, 
					iAdsErrId				=> iAdsErrId, 
					iCANopenErrId			=> iCANopenErrId);
//===============================================================
{endregion}

END_FUNCTION_BLOCK

// ---- POUs/POUsAxisOnline/AX8000/FB_McAxisOnlineAX8000.TcPOU
//==================================================================================================
//							Beckhoff Automation Poland
//									7.12.2018
//	Wszystkomajacy blok funkcyjny do sterowania osia, 
//	wymagane biblioteki: Tc2_EtherCAT, Tc2_MC2_Drive, Tc2_MC2
//  v1.5	|| TC v 3.1.4022.27		|| - dodane opisy bledow w formie zmiennych typu string
// 	v1.4 	|| TC v 3.1.4022.20	 	|| - ACT_MotorMonitoring - only for real axis
// 	v1.3 	|| TC v 3.1.4022.16	 	|| - spojne z AX5000
// 	v1.2 	|| TC v 3.1.4022.16	 	|| - Added ACT_SetPositionIO, migration part of logic from ACT_SetPosition to ACT_SetPositionIO
// 	v1.1 	|| TC v 3.1.4022.16	 	|| - ACT_MotorMonitoring - is executing always, ACT_Initialization - optimalization
// 	v1.0 	|| TC v 3.1.4022.16	 	|| - first edition
//==================================================================================================
{attribute 'reflection'}
FUNCTION_BLOCK FB_McAxisOnlineAX8000
VAR_IN_OUT
	stMcAxisOnline						: ST_McAxisOnline;
	Axis								: AXIS_REF;
END_VAR
VAR
	mcPower								: MC_Power;
	mcStop								: MC_Stop;
	mcHalt								: MC_Halt;
	mcStopSS1							: MC_Stop;
	mcStopSS2							: MC_Stop;
	mcReset								: MC_Reset;
	mcHome								: MC_Home;
	mcSetPosition						: MC_SetPosition;
	fbSetPositionOffset					: FB_CoEAX8000SetPositionOffset;
	mcJog								: MC_Jog;

	mcMoveAbsolute						: MC_MoveAbsolute;
	mcMoveRelative						: MC_MoveRelative;
	mcMoveVelocity						: MC_MoveVelocity;
	mcMoveModulo						: MC_MoveModulo;
	mcMoveAbsolute2						: MC_MoveAbsolute;
	mcMoveRelative2						: MC_MoveRelative;
	mcMoveVelocity2						: MC_MoveVelocity;
	mcMoveModulo2						: MC_MoveModulo;

	fbMotorMonitoring					: FB_MotorMonitoringAX8000;
	fbHoldingBrakeCtrl					: FB_HoldingBrakeCtrlAX8000;
	fbNcLimitSwitch						: FB_NcSWLimitSwitchCtrl;
	tonGetDriveDiag						: TON;
	fbReadChannelErrorCode				: FB_ReadChannelErrorCodeAX8000;
	
	mcReadDriveAddress					: MC_ReadDriveAddress;
	mcReadParameterSet					: MC_ReadParameterSet;
	fbGetDriveRef						: FB_GetDriveRef;

	// Internal
	bInitialized						: BOOL;
	bCommError							: BOOL;
	bReadParameterError					: BOOL;
	bInitError							: BOOL;
	bDriveError							: BOOL;
	bFBError							: BOOL;
	
// Initialization
	iInitStep							: INT;
	bInitializationError				: BOOL;
	wInitializationErrorCounter			: WORD;
	bDriveAddressReady					: BOOL;
	bDriveRefReady						: BOOL;
	bReadParameterSetReady				: BOOL;
	tonDelay							: TON;
// Re init
	udiOnlineChangeCntOld				: UDINT;
	bOnlineChangeDetected				: BOOL;
	bReInit								: BOOL;
	bReInitialized						: BOOL;
	bReInitializationError				: BOOL;
	{attribute 'instance-path'}
	{attribute 'noinit'}
	sInstancePath						: STRING;
END_VAR

// Device dependent initialization 
ACT_Initialization();
// Device independent commands, mostly NC 
ACT_States();
ACT_SWLimitSwitch();
ACT_Stop();
ACT_Power();
ACT_Homing();
ACT_Jog();
ACT_Move();
ACT_Reset();
ACT_SetPosition();
// Device dependent commands
// Motor monitoring possible only with real axis
IF NOT Axis.Status.OpMode.SimulationAxis THEN
	ACT_MotorMonitoring();
END_IF
// Device dependent commands, possible only on real axis after complete initialization
IF bInitialized AND NOT Axis.Status.OpMode.SimulationAxis THEN
	ACT_SetPositionIO();
	ACT_DriveDiag();
	ACT_HoldingBrakeCtrl();
END_IF

// Device independent error collection
ACT_ErrorCollection();

ACTION ACT_DriveDiag:
// Auto update when drive error
tonGetDriveDiag(IN:= stMcAxisOnline.stError.bDriveError AND NOT tonGetDriveDiag.Q, PT:= T#5S, Q=> , ET=> );

fbReadChannelErrorCode(	bExecute				:= stMcAxisOnline.stChannelErrorCode.bExecute OR tonGetDriveDiag.Q,
						stDriveRef				:= stMcAxisOnline.stDriveRef,
						bBusy					=> stMcAxisOnline.stChannelErrorCode.bBusy,
						bError					=> stMcAxisOnline.stChannelErrorCode.bError,
						iAdsErrId				=> stMcAxisOnline.stChannelErrorCode.uiAdsErrId,
						iCANopenErrId			=> stMcAxisOnline.stChannelErrorCode.uiSecErrId,
						uiChannelErrorCode		=> stMcAxisOnline.stChannelErrorCode.uiChannelErrorCode,
						uiChannelErrorCodeHex	=> stMcAxisOnline.stChannelErrorCode.uiChannelErrorCodeHex);
END_ACTION

ACTION ACT_ErrorCollection:
// Error flags
stMcAxisOnline.stError.bDriveError					:= Axis.Status.DriveDeviceError;

stMcAxisOnline.stError.bNcError						:= Axis.Status.Error;

stMcAxisOnline.stError.bFBError						:= stMcAxisOnline.mcPower.bError OR stMcAxisOnline.mcReset.bError OR stMcAxisOnline.mcHome.bError OR stMcAxisOnline.mcJog.bError
													OR stMcAxisOnline.mcHalt.bError OR stMcAxisOnline.mcStop.bError OR stMcAxisOnline.mcSS1.bError OR stMcAxisOnline.mcSS2.bError
													OR stMcAxisOnline.mcMoveAbsolute.bError OR stMcAxisOnline.mcMoveRelative.bError OR stMcAxisOnline.mcMoveVelocity.bError OR stMcAxisOnline.mcMoveModulo.bError
													OR stMcAxisOnline.mcMoveAbsolute2.bError OR stMcAxisOnline.mcMoveRelative2.bError OR stMcAxisOnline.mcMoveVelocity2.bError OR stMcAxisOnline.mcMoveModulo2.bError
													OR stMcAxisOnline.stNcLimitSwitch.bError OR stMcAxisOnline.mcSetPosition.bError;
									
stMcAxisOnline.stError.bCommunicationError			:= stMcAxisOnline.stChannelErrorCode.bError OR stMcAxisOnline.stSetPositionOffset.bError OR stMcAxisOnline.stMotorMonitoring.bError OR stMcAxisOnline.stHoldingBrake.bError;

stMcAxisOnline.stError.bError						:= stMcAxisOnline.stError.bDriveError OR stMcAxisOnline.stError.bNcError OR stMcAxisOnline.stError.bFBError OR stMcAxisOnline.stError.bCommunicationError;
stMcAxisOnline.bError								:= stMcAxisOnline.stError.bError; // Forward one stage up

// Error codes
stMcAxisOnline.stError.uiDriveErrorID 				:= stMcAxisOnline.stChannelErrorCode.uiChannelErrorCode;
stMcAxisOnline.stError.uiDriveErrorIDHex 			:= stMcAxisOnline.stChannelErrorCode.uiChannelErrorCodeHex;

stMcAxisOnline.stError.udiNcErrorID 				:= Axis.Status.ErrorID;
stMcAxisOnline.stError.udiNcErrorIDHex 				:= Axis.Status.ErrorID;
	

stMcAxisOnline.stError.udiFBErrorID 				:= 	stMcAxisOnline.mcPower.udiErrorID + 
														stMcAxisOnline.mcReset.udiErrorID + 
														stMcAxisOnline.mcHome.udiErrorID + 
														stMcAxisOnline.mcJog.udiErrorID +
														stMcAxisOnline.mcHalt.udiErrorID + 
														stMcAxisOnline.mcStop.udiErrorID + 
														stMcAxisOnline.mcSS1.udiErrorID + 
														stMcAxisOnline.mcSS2.udiErrorID +
														stMcAxisOnline.mcMoveAbsolute.udiErrorID + 
														stMcAxisOnline.mcMoveRelative.udiErrorID + 
														stMcAxisOnline.mcMoveVelocity.udiErrorID + 
														stMcAxisOnline.mcMoveModulo.udiErrorID +
														stMcAxisOnline.mcMoveAbsolute2.udiErrorID + 
														stMcAxisOnline.mcMoveRelative2.udiErrorID + 
														stMcAxisOnline.mcMoveVelocity2.udiErrorID + 
														stMcAxisOnline.mcMoveModulo2.udiErrorID +
														stMcAxisOnline.stNcLimitSwitch.udiErrorID + 
														stMcAxisOnline.mcSetPosition.udiErrorID;

stMcAxisOnline.stError.udiFBErrorIDHex 				:= stMcAxisOnline.stError.udiFBErrorID;

stMcAxisOnline.stError.udiErrorID					:= stMcAxisOnline.stSetPositionOffset.udiErrorID;
stMcAxisOnline.stError.uiAdsErrorID					:= stMcAxisOnline.stChannelErrorCode.uiAdsErrId + stMcAxisOnline.stMotorMonitoring.uiAdsErrId + stMcAxisOnline.stHoldingBrake.uiAdsErrId;
stMcAxisOnline.stError.uiSecErrorID					:= stMcAxisOnline.stChannelErrorCode.uiSecErrId + stMcAxisOnline.stMotorMonitoring.uiSecErrId + stMcAxisOnline.stHoldingBrake.uiSecErrId;

stMcAxisOnline.stError.sNcError						:= F_AxErrMsg(stMcAxisOnline.stError.udiNcErrorID);
stMcAxisOnline.stError.sDriveError					:= F_AX8xErrMsg(stMcAxisOnline.stError.uiDriveErrorID);
END_ACTION

ACTION ACT_HoldingBrakeCtrl:
fbHoldingBrakeCtrl(	bForceLock			:= stMcAxisOnline.stHoldingBrake.bForceLock,
					bForceUnlock		:= stMcAxisOnline.stHoldingBrake.bForceUnlock,
					stDriveRef			:= stMcAxisOnline.stDriveRef,
					bBusy				=> stMcAxisOnline.stHoldingBrake.bBusy,
					bError				=> stMcAxisOnline.stHoldingBrake.bError,
					iAdsErrId			=> stMcAxisOnline.stHoldingBrake.uiAdsErrId,
					iCANopenErrId		=> stMcAxisOnline.stHoldingBrake.uiSecErrId);
END_ACTION

ACTION ACT_Homing:
mcHome(		Axis						:= Axis,
			Execute						:= stMcAxisOnline.mcHome.bExecute,
			Position					:= stMcAxisOnline.mcHome.lrPosition,
			HomingMode					:= stMcAxisOnline.mcHome.eHomingMode,
			BufferMode					:= stMcAxisOnline.mcHome.eBufferMode,
			Options						:= stMcAxisOnline.mcHome.stOptions,
			bCalibrationCam				:= stMcAxisOnline.mcHome.bCalibrationCam,
			Done						=> stMcAxisOnline.mcHome.bDone,
			Busy						=> stMcAxisOnline.mcHome.bBusy,
			Active						=> stMcAxisOnline.mcHome.bActive,
			CommandAborted				=> stMcAxisOnline.mcHome.bCommandAborted,
			Error						=> stMcAxisOnline.mcHome.bError,
			ErrorID						=> stMcAxisOnline.mcHome.udiErrorID);
END_ACTION

ACTION ACT_Initialization:
// bInitialized flag is set just once. 
// bReInitialized ise set each time we do online change or request reinit operation
// bDriveAddressReady, bReadParameterSetReady, bDriveRefReady - set just once after successed read

// Online change detection
bOnlineChangeDetected					:= udiOnlineChangeCntOld <> _AppInfo.OnlineChangeCnt;
udiOnlineChangeCntOld 					:= _AppInfo.OnlineChangeCnt;
// Reset init
IF bReInit OR bOnlineChangeDetected THEN
	iInitStep							:= 0;
END_IF

//Initialization process
CASE iInitStep OF
	0:	// Read Drive Address
		
		stMcAxisOnline.mcReadDriveAddress.bExecute	:=	 TRUE;
		iInitStep						:= iInitStep + 10;
		
	10: // Wait for data
	
		IF NOT stMcAxisOnline.mcReadDriveAddress.bBusy THEN
			stMcAxisOnline.mcReadDriveAddress.bExecute	:=	 FALSE;
			IF stMcAxisOnline.mcReadDriveAddress.bDone THEN
				iInitStep 				:= iInitStep + 10;
				bDriveAddressReady 		:= TRUE;
			ELSE
				iInitStep 				:= 1000;		// Error step
			END_IF
		END_IF
		
	20:	// Read Parameter Set
		
		stMcAxisOnline.mcReadParameterSet.bExecute		:=	 TRUE;
		iInitStep						:= iInitStep + 10;
		
	30: // Wait for data
	
		IF NOT stMcAxisOnline.mcReadParameterSet.bBusy THEN
			stMcAxisOnline.mcReadParameterSet.bExecute	:=	 FALSE;
			IF stMcAxisOnline.mcReadParameterSet.bDone THEN
				iInitStep 				:= iInitStep + 10;
				bReadParameterSetReady 	:= TRUE;
			ELSE
				iInitStep 				:= 1000;		// Error step
			END_IF
		END_IF	
	
	40:	// Get Drive Ref
		
		stMcAxisOnline.stGetDriveRef.bExecute		:=	 TRUE;
		iInitStep						:= iInitStep + 10;
		
	50: // Wait for data
	
		IF NOT stMcAxisOnline.stGetDriveRef.bBusy THEN
			stMcAxisOnline.stGetDriveRef.bExecute	:=	 FALSE;
			IF NOT stMcAxisOnline.stGetDriveRef.bError THEN
				iInitStep 				:= iInitStep + 10;
				bDriveRefReady 			:= TRUE;
			ELSE
				iInitStep 				:= 1000;		// Error step
			END_IF
		END_IF
	
	60: // Success - initialized flag, clear error
		bReInitialized					:= bInitialized;	// TRUE only when it's not first initialization e.g. online change
		bInitialized 					:= TRUE;
		bReInitializationError			:= FALSE;			// TRUE only when it's not first initialization e.g. online change
		bInitializationError			:= FALSE;
		iInitStep 						:= iInitStep + 10;
		
	70: // Idle
	
		;
		
	1000: // Error step
		wInitializationErrorCounter 	:= wInitializationErrorCounter + 1;
		IF wInitializationErrorCounter < 100 THEN
			iInitStep					:= iInitStep + 5;			// Go to delay
		ELSE
			bReInitializationError		:= bInitializationError;	// TRUE only when it's not first initialization e.g. online change
			bInitializationError		:= TRUE;
			bReInitialized				:= FALSE;
			iInitStep 					:= iInitStep + 10;
		END_IF

	1005: // Delay step
		tonDelay(IN:= TRUE, PT:= T#1S);
		IF tonDelay.Q THEN
			tonDelay(IN:= FALSE, PT:= T#1S);
			iInitStep					:= 0;
		END_IF
		
	1010: // Idle after error
		;
	
END_CASE

mcReadDriveAddress(	Axis				:= Axis,
					Execute				:= stMcAxisOnline.mcReadDriveAddress.bExecute,
					Done				=> stMcAxisOnline.mcReadDriveAddress.bDone,
					Busy				=> stMcAxisOnline.mcReadDriveAddress.bBusy,
					Error				=> stMcAxisOnline.mcReadDriveAddress.bError,
					ErrorID				=> stMcAxisOnline.mcReadDriveAddress.udiErrorID,
					DriveAddress		=> stMcAxisOnline.stDriveAddress);
				
mcReadParameterSet(	Parameter			:= stMcAxisOnline.stAxisParameter,
					Axis				:= Axis,
					Execute				:= stMcAxisOnline.mcReadParameterSet.bExecute,
					Done				=> stMcAxisOnline.mcReadParameterSet.bDone,
					Busy				=> stMcAxisOnline.mcReadParameterSet.bBusy,
					Error				=> stMcAxisOnline.mcReadParameterSet.bError,
					ErrorID				=> stMcAxisOnline.mcReadParameterSet.udiErrorID);
					
fbGetDriveRef(		bExecute			:= stMcAxisOnline.stGetDriveRef.bExecute,
					bBusy				=> stMcAxisOnline.stGetDriveRef.bBusy,
					bError				=> stMcAxisOnline.stGetDriveRef.bError,
					udiErrorID			=> stMcAxisOnline.stGetDriveRef.udiErrorID,
					stDriveRef			=> stMcAxisOnline.stDriveRef,
					Axis				:= Axis);
END_ACTION

ACTION ACT_Jog:
// Direct access from bSlow or bFast, if none then free choice
IF stMcAxisOnline.mcJog.bSlowForward OR stMcAxisOnline.mcJog.bSlowBackward THEN
	stMcAxisOnline.mcJog.eMode			:= MC_JOGMODE_STANDARD_SLOW;
ELSIF stMcAxisOnline.mcJog.bFastForward OR stMcAxisOnline.mcJog.bFastBackward THEN
	stMcAxisOnline.mcJog.eMode			:= MC_JOGMODE_STANDARD_FAST;
END_IF

mcJog(		Axis						:= Axis,
			JogForward					:= stMcAxisOnline.mcJog.bJogForward OR stMcAxisOnline.mcJog.bSlowForward OR stMcAxisOnline.mcJog.bFastForward,
			JogBackwards				:= stMcAxisOnline.mcJog.bJogBackwards OR stMcAxisOnline.mcJog.bSlowBackward OR stMcAxisOnline.mcJog.bFastBackward,
			Mode						:= stMcAxisOnline.mcJog.eMode,
			Position					:= stMcAxisOnline.mcJog.lrPosition,
			Velocity					:= stMcAxisOnline.mcJog.lrVelocity,
			Acceleration				:= stMcAxisOnline.mcJog.lrAcceleration,
			Deceleration				:= stMcAxisOnline.mcJog.lrDeceleration,
			Jerk						:= stMcAxisOnline.mcJog.lrJerk,
			Done						=> stMcAxisOnline.mcJog.bDone,
			Busy						=> stMcAxisOnline.mcJog.bBusy,
			Active						=> stMcAxisOnline.mcJog.bActive,
			CommandAborted				=> stMcAxisOnline.mcJog.bCommandAborted,
			Error						=> stMcAxisOnline.mcJog.bError,
			ErrorID						=> stMcAxisOnline.mcJog.udiErrorID);
END_ACTION

ACTION ACT_MotorMonitoring:
fbMotorMonitoring(	bReset				:= stMcAxisOnline.stMotorMonitoring.bReset,
					rTorqueLimit		:= stMcAxisOnline.stMotorMonitoring.rTorqueLimit,
					stDriveRef			:= stMcAxisOnline.stDriveRef,
					bError				=> stMcAxisOnline.stMotorMonitoring.bError,
					uiAdsErrId			=> stMcAxisOnline.stMotorMonitoring.uiAdsErrId,
					uiCANopenErrId		=> stMcAxisOnline.stMotorMonitoring.uiSecErrId,
					bInitialized		=> stMcAxisOnline.stMotorMonitoring.bInitialized,
					bWarning			=> stMcAxisOnline.stMotorMonitoring.bWarning,
					rWarningCurrent		=> stMcAxisOnline.stMotorMonitoring.rWarningCurrent,
					rTorquePerc			=> stMcAxisOnline.stMotorMonitoring.rTorquePerc,
					rTorquePercMax		=> stMcAxisOnline.stMotorMonitoring.rTorquePercMax,
					rTorque				=> stMcAxisOnline.stMotorMonitoring.rTorque,
					rTorqueF			=> stMcAxisOnline.stMotorMonitoring.rTorqueF,
					rTorqueMax			=> stMcAxisOnline.stMotorMonitoring.rTorqueMax,
					rCurrent			=> stMcAxisOnline.stMotorMonitoring.rCurrent,
					rCurrentF			=> stMcAxisOnline.stMotorMonitoring.rCurrentF,
					rCurrentMax			=> stMcAxisOnline.stMotorMonitoring.rCurrentMax,
					rI2T				=> stMcAxisOnline.stMotorMonitoring.rI2T,
					rI2TMax				=> stMcAxisOnline.stMotorMonitoring.rI2TMax,
					Axis				:= Axis);
END_ACTION

ACTION ACT_Move:
{region "Primary"}
mcMoveAbsolute(	Axis					:= Axis,
				Execute					:= stMcAxisOnline.mcMoveAbsolute.bExecute,
				Position				:= stMcAxisOnline.mcMoveAbsolute.lrPosition,
				Velocity				:= stMcAxisOnline.mcMoveAbsolute.lrVelocity,
				Acceleration			:= stMcAxisOnline.mcMoveAbsolute.lrAcceleration,
				Deceleration			:= stMcAxisOnline.mcMoveAbsolute.lrDeceleration,
				Jerk					:= stMcAxisOnline.mcMoveAbsolute.lrJerk,
				BufferMode				:= stMcAxisOnline.mcMoveAbsolute.eBufferMode,
				Options					:= stMcAxisOnline.mcMoveAbsolute.stOptions,
				Done					=> stMcAxisOnline.mcMoveAbsolute.bDone,
				Busy					=> stMcAxisOnline.mcMoveAbsolute.bBusy,
				Active					=> stMcAxisOnline.mcMoveAbsolute.bActive,
				CommandAborted			=> stMcAxisOnline.mcMoveAbsolute.bCommandAborted,
				Error					=> stMcAxisOnline.mcMoveAbsolute.bError,
				ErrorID					=> stMcAxisOnline.mcMoveAbsolute.udiErrorID);

mcMoveRelative(	Axis					:= Axis,
				Execute					:= stMcAxisOnline.mcMoveRelative.bExecute,
				Distance				:= stMcAxisOnline.mcMoveRelative.lrDistance,
				Velocity				:= stMcAxisOnline.mcMoveRelative.lrVelocity,
				Acceleration			:= stMcAxisOnline.mcMoveRelative.lrAcceleration,
				Deceleration			:= stMcAxisOnline.mcMoveRelative.lrDeceleration,
				Jerk					:= stMcAxisOnline.mcMoveRelative.lrJerk,
				BufferMode				:= stMcAxisOnline.mcMoveRelative.eBufferMode,
				Options					:= stMcAxisOnline.mcMoveRelative.stOptions,
				Done					=> stMcAxisOnline.mcMoveRelative.bDone,
				Busy					=> stMcAxisOnline.mcMoveRelative.bBusy,
				Active					=> stMcAxisOnline.mcMoveRelative.bActive,
				CommandAborted			=> stMcAxisOnline.mcMoveRelative.bCommandAborted,
				Error					=> stMcAxisOnline.mcMoveRelative.bError,
				ErrorID					=> stMcAxisOnline.mcMoveRelative.udiErrorID);
				
mcMoveVelocity(	Axis					:= Axis,
				Execute					:= stMcAxisOnline.mcMoveVelocity.bExecute,
				Velocity				:= stMcAxisOnline.mcMoveVelocity.lrVelocity,
				Acceleration			:= stMcAxisOnline.mcMoveVelocity.lrAcceleration,
				Deceleration			:= stMcAxisOnline.mcMoveVelocity.lrDeceleration,
				Jerk					:= stMcAxisOnline.mcMoveVelocity.lrJerk,
				Direction				:= stMcAxisOnline.mcMoveVelocity.eDirection,
				BufferMode				:= stMcAxisOnline.mcMoveVelocity.eBufferMode,
				Options					:= stMcAxisOnline.mcMoveVelocity.stOptions,
				InVelocity				=> stMcAxisOnline.mcMoveVelocity.bInVelocity,
				Busy					=> stMcAxisOnline.mcMoveVelocity.bBusy,
				Active					=> stMcAxisOnline.mcMoveVelocity.bActive,
				CommandAborted			=> stMcAxisOnline.mcMoveVelocity.bCommandAborted,
				Error					=> stMcAxisOnline.mcMoveVelocity.bError,
				ErrorID					=> stMcAxisOnline.mcMoveVelocity.udiErrorID);
stMcAxisOnline.mcMoveVelocity.bDone		:= stMcAxisOnline.mcMoveVelocity.bInVelocity;

mcMoveModulo(	Axis					:= Axis,
				Execute					:= stMcAxisOnline.mcMoveModulo.bExecute,
				Position				:= stMcAxisOnline.mcMoveModulo.lrPosition,
				Velocity				:= stMcAxisOnline.mcMoveModulo.lrVelocity,
				Acceleration			:= stMcAxisOnline.mcMoveModulo.lrAcceleration,
				Deceleration			:= stMcAxisOnline.mcMoveModulo.lrDeceleration,
				Jerk					:= stMcAxisOnline.mcMoveModulo.lrJerk,
				Direction				:= stMcAxisOnline.mcMoveModulo.eDirection,
				BufferMode				:= stMcAxisOnline.mcMoveModulo.eBufferMode,
				Options					:= stMcAxisOnline.mcMoveModulo.stOptions,
				Done					=> stMcAxisOnline.mcMoveModulo.bDone,
				Busy					=> stMcAxisOnline.mcMoveModulo.bBusy,
				Active					=> stMcAxisOnline.mcMoveModulo.bActive,
				CommandAborted			=> stMcAxisOnline.mcMoveModulo.bCommandAborted,
				Error					=> stMcAxisOnline.mcMoveModulo.bError,
				ErrorID					=> stMcAxisOnline.mcMoveModulo.udiErrorID);
{endregion}
{region "Secondary"}
mcMoveAbsolute2(Axis					:= Axis,
				Execute					:= stMcAxisOnline.mcMoveAbsolute2.bExecute,
				Position				:= stMcAxisOnline.mcMoveAbsolute2.lrPosition,
				Velocity				:= stMcAxisOnline.mcMoveAbsolute2.lrVelocity,
				Acceleration			:= stMcAxisOnline.mcMoveAbsolute2.lrAcceleration,
				Deceleration			:= stMcAxisOnline.mcMoveAbsolute2.lrDeceleration,
				Jerk					:= stMcAxisOnline.mcMoveAbsolute2.lrJerk,
				BufferMode				:= stMcAxisOnline.mcMoveAbsolute2.eBufferMode,
				Options					:= stMcAxisOnline.mcMoveAbsolute2.stOptions,
				Done					=> stMcAxisOnline.mcMoveAbsolute2.bDone,
				Busy					=> stMcAxisOnline.mcMoveAbsolute2.bBusy,
				Active					=> stMcAxisOnline.mcMoveAbsolute2.bActive,
				CommandAborted			=> stMcAxisOnline.mcMoveAbsolute2.bCommandAborted,
				Error					=> stMcAxisOnline.mcMoveAbsolute2.bError,
				ErrorID					=> stMcAxisOnline.mcMoveAbsolute2.udiErrorID);

mcMoveRelative2(Axis					:= Axis,
				Execute					:= stMcAxisOnline.mcMoveRelative2.bExecute,
				Distance				:= stMcAxisOnline.mcMoveRelative2.lrDistance,
				Velocity				:= stMcAxisOnline.mcMoveRelative2.lrVelocity,
				Acceleration			:= stMcAxisOnline.mcMoveRelative2.lrAcceleration,
				Deceleration			:= stMcAxisOnline.mcMoveRelative2.lrDeceleration,
				Jerk					:= stMcAxisOnline.mcMoveRelative2.lrJerk,
				BufferMode				:= stMcAxisOnline.mcMoveRelative2.eBufferMode,
				Options					:= stMcAxisOnline.mcMoveRelative2.stOptions,
				Done					=> stMcAxisOnline.mcMoveRelative2.bDone,
				Busy					=> stMcAxisOnline.mcMoveRelative2.bBusy,
				Active					=> stMcAxisOnline.mcMoveRelative2.bActive,
				CommandAborted			=> stMcAxisOnline.mcMoveRelative2.bCommandAborted,
				Error					=> stMcAxisOnline.mcMoveRelative2.bError,
				ErrorID					=> stMcAxisOnline.mcMoveRelative2.udiErrorID);
				
mcMoveVelocity2(Axis					:= Axis,
				Execute					:= stMcAxisOnline.mcMoveVelocity2.bExecute,
				Velocity				:= stMcAxisOnline.mcMoveVelocity2.lrVelocity,
				Acceleration			:= stMcAxisOnline.mcMoveVelocity2.lrAcceleration,
				Deceleration			:= stMcAxisOnline.mcMoveVelocity2.lrDeceleration,
				Jerk					:= stMcAxisOnline.mcMoveVelocity2.lrJerk,
				Direction				:= stMcAxisOnline.mcMoveVelocity2.eDirection,
				BufferMode				:= stMcAxisOnline.mcMoveVelocity2.eBufferMode,
				Options					:= stMcAxisOnline.mcMoveVelocity2.stOptions,
				InVelocity				=> stMcAxisOnline.mcMoveVelocity2.bInVelocity,
				Busy					=> stMcAxisOnline.mcMoveVelocity2.bBusy,
				Active					=> stMcAxisOnline.mcMoveVelocity2.bActive,
				CommandAborted			=> stMcAxisOnline.mcMoveVelocity2.bCommandAborted,
				Error					=> stMcAxisOnline.mcMoveVelocity2.bError,
				ErrorID					=> stMcAxisOnline.mcMoveVelocity2.udiErrorID);
stMcAxisOnline.mcMoveVelocity2.bDone	:= stMcAxisOnline.mcMoveVelocity2.bInVelocity;

mcMoveModulo2(	Axis					:= Axis,
				Execute					:= stMcAxisOnline.mcMoveModulo2.bExecute,
				Position				:= stMcAxisOnline.mcMoveModulo2.lrPosition,
				Velocity				:= stMcAxisOnline.mcMoveModulo2.lrVelocity,
				Acceleration			:= stMcAxisOnline.mcMoveModulo2.lrAcceleration,
				Deceleration			:= stMcAxisOnline.mcMoveModulo2.lrDeceleration,
				Jerk					:= stMcAxisOnline.mcMoveModulo2.lrJerk,
				Direction				:= stMcAxisOnline.mcMoveModulo2.eDirection,
				BufferMode				:= stMcAxisOnline.mcMoveModulo2.eBufferMode,
				Options					:= stMcAxisOnline.mcMoveModulo2.stOptions,
				Done					=> stMcAxisOnline.mcMoveModulo2.bDone,
				Busy					=> stMcAxisOnline.mcMoveModulo2.bBusy,
				Active					=> stMcAxisOnline.mcMoveModulo2.bActive,
				CommandAborted			=> stMcAxisOnline.mcMoveModulo2.bCommandAborted,
				Error					=> stMcAxisOnline.mcMoveModulo2.bError,
				ErrorID					=> stMcAxisOnline.mcMoveModulo2.udiErrorID);
{endregion}
END_ACTION

ACTION ACT_Power:
mcPower(	Axis						:= Axis,									//
			Enable						:= stMcAxisOnline.mcPower.bEnable,
			Enable_Positive				:= stMcAxisOnline.mcPower.bEnable_Positive,
			Enable_Negative				:= stMcAxisOnline.mcPower.bEnable_Negative,
			Override					:= stMcAxisOnline.mcPower.lrOverride,
			BufferMode					:= stMcAxisOnline.mcPower.eBufferMode,
			Options						:= stMcAxisOnline.mcPower.stOptions,
			Status						=> stMcAxisOnline.mcPower.bStatus,
			Busy						=> stMcAxisOnline.mcPower.bBusy,
			Active						=> stMcAxisOnline.mcPower.bActive,
			Error						=> stMcAxisOnline.mcPower.bError,
			ErrorID						=> stMcAxisOnline.mcPower.udiErrorID);
END_ACTION

ACTION ACT_Reset:
mcReset(	Axis						:= Axis,
			Execute						:= stMcAxisOnline.mcReset.bExecute,
			Done						=> stMcAxisOnline.mcReset.bDone,
			Busy						=> stMcAxisOnline.mcReset.bBusy,
			Error						=> stMcAxisOnline.mcReset.bError,
			ErrorID						=> stMcAxisOnline.mcReset.udiErrorID);
END_ACTION

ACTION ACT_SetPosition:
mcSetPosition(		Axis				:= Axis,
					Execute				:= stMcAxisOnline.mcSetPosition.bExecute,
					Position			:= stMcAxisOnline.mcSetPosition.lrPosition,
					Mode				:= stMcAxisOnline.mcSetPosition.bMode,
					Options				:= stMcAxisOnline.mcSetPosition.stOptions,
					Done				=> stMcAxisOnline.mcSetPosition.bDone,
					Busy				=> stMcAxisOnline.mcSetPosition.bBusy,
					Error				=> stMcAxisOnline.mcSetPosition.bError,
					ErrorID				=> stMcAxisOnline.mcSetPosition.udiErrorID);
END_ACTION

ACTION ACT_SetPositionIO:
fbSetPositionOffset(Execute				:= stMcAxisOnline.stSetPositionOffset.bExecute,
					Position			:= stMcAxisOnline.stSetPositionOffset.lrPosition,
					Relative			:= stMcAxisOnline.stSetPositionOffset.bRelative,
					Feedback			:= stMcAxisOnline.stSetPositionOffset.eFeedback,
					Memory				:= stMcAxisOnline.stSetPositionOffset.eMemory,
					Busy				=> stMcAxisOnline.stSetPositionOffset.bBusy,
					Error				=> stMcAxisOnline.stSetPositionOffset.bError,
					ErrorID				=> stMcAxisOnline.stSetPositionOffset.udiErrorID,
					Axis				:= Axis);
END_ACTION

ACTION ACT_States:
// Read States and forward main states
Axis.ReadStatus();
stMcAxisOnline.stStatus.stAxisStatus		:= Axis.Status;
stMcAxisOnline.stStatus.dwAxisId			:= Axis.NcToPlc.AxisId;
stMcAxisOnline.stStatus.bNcError			:= Axis.Status.Error;
stMcAxisOnline.stStatus.udiNcErrorCode		:= Axis.Status.ErrorID;
stMcAxisOnline.stStatus.udiNcErrorCodeHex	:= Axis.Status.ErrorID;

stMcAxisOnline.stStatus.sAxisName			:= stMcAxisOnline.stAxisParameter.sAxisName;
stMcAxisOnline.stStatus.lrActPos			:= Axis.NcToPlc.ActPos;
stMcAxisOnline.stStatus.lrModuloActPos		:= Axis.NcToPlc.ModuloActPos;
stMcAxisOnline.stStatus.lrActVelo			:= Axis.NcToPlc.ActVelo;
stMcAxisOnline.stStatus.lrActAcc			:= Axis.NcToPlc.ActAcc;
stMcAxisOnline.stStatus.lrActTorque			:= Axis.NcToPlc.ActTorque;
stMcAxisOnline.stStatus.lrPosDiff			:= Axis.NcToPlc.PosDiff;
stMcAxisOnline.stStatus.lrSetPos			:= Axis.NcToPlc.SetPos;
stMcAxisOnline.stStatus.lrSetVelo			:= Axis.NcToPlc.SetVelo;
stMcAxisOnline.stStatus.lrSetAcc			:= Axis.NcToPlc.SetAcc;
stMcAxisOnline.stStatus.lrSetTorque			:= Axis.NcToPlc.SetTorque;
stMcAxisOnline.stStatus.lrPosDiff			:= Axis.NcToPlc.PosDiff;
stMcAxisOnline.stStatus.bAxisReady			:= Axis.Status.Operational;
stMcAxisOnline.stStatus.bHomed				:= Axis.Status.Homed;
stMcAxisOnline.stStatus.bCoupled			:= Axis.Status.Coupled;

// zezwolenie na zjazd z krancowki hw
Axis.PlcToNc.ControlDWord.8				:= stMcAxisOnline.stStatus.bAcceptBlockedDrive;
END_ACTION

ACTION ACT_Stop:
mcHalt(		Axis						:= Axis,
			Execute						:= stMcAxisOnline.mcHalt.bExecute,
			Deceleration				:= stMcAxisOnline.mcHalt.lrDeceleration,
			Jerk						:= stMcAxisOnline.mcHalt.lrJerk,
			BufferMode					:= stMcAxisOnline.mcHalt.eBufferMode,
			Options						:= stMcAxisOnline.mcHalt.stOptions,
			Done						=> stMcAxisOnline.mcHalt.bDone,
			Busy						=> stMcAxisOnline.mcHalt.bBusy,
			Active						=> stMcAxisOnline.mcHalt.bActive,
			CommandAborted				=> stMcAxisOnline.mcHalt.bCommandAborted,
			Error						=> stMcAxisOnline.mcHalt.bError,
			ErrorID						=> stMcAxisOnline.mcHalt.udiErrorID);
			
mcStop(		Axis						:= Axis,
			Execute						:= stMcAxisOnline.mcStop.bExecute,
			Deceleration				:= stMcAxisOnline.mcStop.lrDeceleration,
			Jerk						:= stMcAxisOnline.mcStop.lrJerk,
			Options						:= stMcAxisOnline.mcStop.stOptions,
			Done						=> stMcAxisOnline.mcStop.bDone,
			Busy						=> stMcAxisOnline.mcStop.bBusy,
			Active						=> stMcAxisOnline.mcStop.bActive,
			CommandAborted				=> stMcAxisOnline.mcStop.bCommandAborted,
			Error						=> stMcAxisOnline.mcStop.bError,
			ErrorID						=> stMcAxisOnline.mcStop.udiErrorID);
			
mcStopSS2(	Axis						:= Axis,
			Execute						:= stMcAxisOnline.mcSS2.bExecute,
			Deceleration				:= stMcAxisOnline.mcSS2.lrDeceleration,
			Jerk						:= stMcAxisOnline.mcSS2.lrJerk,
			Options						:= stMcAxisOnline.mcSS2.stOptions,
			Done						=> stMcAxisOnline.mcSS2.bDone,
			Busy						=> stMcAxisOnline.mcSS2.bBusy,
			Active						=> stMcAxisOnline.mcSS2.bActive,
			CommandAborted				=> stMcAxisOnline.mcSS2.bCommandAborted,
			Error						=> stMcAxisOnline.mcSS2.bError,
			ErrorID						=> stMcAxisOnline.mcSS2.udiErrorID);
			
mcStopSS1(	Axis						:= Axis,
			Execute						:= stMcAxisOnline.mcSS1.bExecute,
			Deceleration				:= stMcAxisOnline.mcSS1.lrDeceleration,
			Jerk						:= stMcAxisOnline.mcSS1.lrJerk,
			Options						:= stMcAxisOnline.mcSS1.stOptions,
			Done						=> stMcAxisOnline.mcSS1.bDone,
			Busy						=> stMcAxisOnline.mcSS1.bBusy,
			Active						=> stMcAxisOnline.mcSS1.bActive,
			CommandAborted				=> stMcAxisOnline.mcSS1.bCommandAborted,
			Error						=> stMcAxisOnline.mcSS1.bError,
			ErrorID						=> stMcAxisOnline.mcSS1.udiErrorID);
// SS1 - after MC_Stop function we have to disable drive			
stMcAxisOnline.mcPower.bEnable R= stMcAxisOnline.mcPower.bEnable_Positive R= stMcAxisOnline.mcPower.bEnable_Negative R= (stMcAxisOnline.mcSS1.bDone OR stMcAxisOnline.mcSS1.bCommandAborted OR stMcAxisOnline.mcSS1.bError);
END_ACTION

ACTION ACT_SWLimitSwitch:
fbNcLimitSwitch(	udiAxisID		:= Axis.NcToPlc.AxisId, 
					bRead			:= stMcAxisOnline.stNcLimitSwitch.bRead, 
					bWrite			:= stMcAxisOnline.stNcLimitSwitch.bWrite, 
					bReset			:= stMcAxisOnline.stNcLimitSwitch.bReset, 
					lrSetMinPos		:= stMcAxisOnline.stNcLimitSwitch.lrSetMinPos, 
					lrSetMaxPos		:= stMcAxisOnline.stNcLimitSwitch.lrSetMaxPos, 
					bSetMinMon		:= stMcAxisOnline.stNcLimitSwitch.bSetMinMon, 
					bSetMaxMon		:= stMcAxisOnline.stNcLimitSwitch.bSetMaxMon, 
					bBusy			=> stMcAxisOnline.stNcLimitSwitch.bBusy, 
					bError			=> stMcAxisOnline.stNcLimitSwitch.bError, 
					udiErrorID		=> stMcAxisOnline.stNcLimitSwitch.udiErrorID, 
					lrActMinPos		=> stMcAxisOnline.stNcLimitSwitch.lrActMinPos, 
					lrActMaxPos		=> stMcAxisOnline.stNcLimitSwitch.lrActMaxPos, 
					bActMinMon		=> stMcAxisOnline.stNcLimitSwitch.bActMinMon, 
					bActMaxMon		=> stMcAxisOnline.stNcLimitSwitch.bActMaxMon);
END_ACTION

END_FUNCTION_BLOCK

// ---- POUs/POUsAxisOnline/AX8000/FB_MotorMonitoringAX8000.TcPOU
//==================================================================================================
//							Beckhoff Automation Poland
//									4.07.2018
//	Blok funkcyjny pozwala na monitorowanie i ograniczanie momentu oraz monitoring parametru I2T dla AX8xxx.
//	Zmienne do zlinkowania zadeklarowane są wewnątrz bloku.
//	Ograniczenie i monitorowanie momentu
//	Ograniczenie momentu podawane jest przez wejście rTorqueLimit.
//	Na wyjściu podana jest wartość surowa w %, jak i przeskalowana na A (prąd) i Nm (moment).
//	Blok zwraca wartości bieżące, przefiltrowane i maksymalne.
//	Wartości maksymalne mogą być wyzerowane za pomocą zmiennej bReset.
//	Wewnętrznie wykorzystany jest blok FB_FilterEx.
//
//  v1.3	|| TC v 3.1.4022.22		|| - reset na poczatku bloku, optymalizacja kodu
//  v1.2	|| TC v 3.1.4022.16		|| - inicjalizacja po 10 nieudanych probach zglasza blad
//  v1.1	|| TC v 3.1.4022.16		|| - wyjscie iTorque przeniesione do lokalnych, w jego miejsce rTorquePerc i rTorquePercMax, 
//										flaga bTorqueLimitOK zalezna tylko od rTorqueLimitLow, zmiana nazw zgodnie z typami: uiAdsErrId, uiCANopenErrId
//  v1.0	|| TC v 3.1.4022.16		|| - pierwsza wersja
//==================================================================================================
FUNCTION_BLOCK FB_MotorMonitoringAX8000
VAR CONSTANT
	rTorqueLimitLow					: REAL 		:= 0.01;				// Low limit used for bipolar torque limit value
	rTorqueLimitHigh				: REAL		:= 500.0;				// High limit used for bipolar torque limit value
END_VAR
VAR_INPUT
	bReset							: BOOL;								// Reset FB
	rTorqueLimit					: REAL 		:= rTorqueLimitHigh; 	// Bipolar torque limit: 0-500%, resolution 0.1%, value goes to: 16#6072 (Ch A)/ 16#6872 (Ch B)
	stDriveRef						: ST_DriveRef;						// Necessary for FB_CoERead_ByDriveRef
END_VAR
VAR_OUTPUT
	bError							: BOOL; 							// General error: parameter or CoE read.
																		// If bError = TRUE and bInitialized = FALSE - error during read motor data.
																		// If bError = TRUE and bInitialized = TRUE and (iAdsErrId <> 0 or iCANopenErrId <> 0) then I2T read error
																		// If bError = TRUE and bInitialized = TRUE and iAdsErrId = 0 and iCANopenErrId = 0 then parameter error: rTorqueLimit outside permitted range rTorqueLimitLow..rTorqueLimitHigh or Empty stDriveRef
	uiAdsErrId						: UINT;								// Forwarded output FB_CoERead_ByDriveRef
	uiCANopenErrId					: UINT;								// Forwarded output FB_CoERead_ByDriveRef
	bInitialized					: BOOL;								// TRUE - Motor data read without errors, so it's possible to calculate torqe and current values in metric units
	bWarning						: BOOL;								// rCurrentF > rWarningCurrent, be aware to be over permitted range
	rWarningCurrent					: REAL; 							// Continuous Stall Current - motor parameter: 16#6075 (Ch A)/ 16#6875 (Ch B); scalled: [A]
	rTorquePerc						: REAL;								// [%]
	rTorquePercMax					: REAL;								// Max [%]
	rTorque							: REAL; 							// [Nm]
	rTorqueF						: REAL;								// Filtered [Nm]
	rTorqueMax						: REAL;								// Max [Nm]
	rCurrent						: REAL; 							// [A]
	rCurrentF						: REAL;								// Filtered [A]
	rCurrentMax						: REAL;								// Max [A]
	rI2T							: REAL; 							// Thermal Motor Utilization: 16#32C1:02 (Ch A)/ 16#36C1:02 (Ch B); units: [%]
	rI2TMax							: REAL; 							// Max % Nominal
END_VAR
VAR_IN_OUT
	Axis							: AXIS_REF;							// Axis Ref struct
END_VAR
VAR
//======================= Internal var ===========================
	iStep							: INT;								// Case instruction
	bDriveRefOK						: BOOL;								// stDriveRef contains necessary data to read CoE
	bTorqueLimitOK					: BOOL;								// rTorqueLimit in permitted range rTorqueLimitLow..rTorqueLimitHigh
	uiBipolarTorqueLimitValue  		AT %Q*: UINT; 						// Raw data, linked to Bipolar torque limit value
	iTorque 						: INT; 								// -1000 .. 1000 - RAW values the same as process image
	rTorqueRAW						: REAL; 							// -1000 .. 1000 - RAW values the same as process image
	rSfTorque						: REAL; 							// RAW -1000..1000 --> Nm
	rSfCurrent						: REAL; 							// Nm --> A
	udiMotorStandstillCurrent		: UDINT;							// 16#6075 (Ch A)/ 16#6875 (Ch B); units: [mA]
	udiMotorStandstillTorque		: UDINT;							// 16#6076 (Ch A)/ 16#6876 (Ch B); units: [mNm]
	wInitErrorCount					: WORD;								// Initialization error counter, if bigger then 10 then error
//========================== FBs ================================
	rtReset							: R_TRIG;							// Reset trigger
	tonWait							: TON;								// Wait timer - used for I2T read interval and for repeat initialization
	fbFilterEx						: FB_FilterEx;						// Filter
	fbCoERead						: FB_CoERead_ByDriveRef;			// FB for read CoE parameters
//===============================================================
END_VAR

//============== Reset max values and FB ========================
rtReset(CLK:= bReset);
IF rtReset.Q THEN
	fbCoERead.bExecute					:= FALSE;
	rCurrentMax							:= 0;
	rTorqueMax 							:= 0;
	rI2TMax								:= 0;
	uiAdsErrId		 					:= 0;
	uiCANopenErrId	 					:= 0;
	iStep								:= 0;
	wInitErrorCount						:= 0;
END_IF
//=================== Call triggers and timers ==================
tonWait(IN:= NOT tonWait.Q, PT:= T#1S);
//======= Check for parameter error - each cycle ================
bDriveRefOK 							:= (stDriveRef.nSlaveAddr <> 0) AND (stDriveRef.sNetId <> '');
bTorqueLimitOK 							:= (rTorqueLimit > rTorqueLimitLow);
//============= Read params and calculations ====================
CASE iStep OF
	
	0: // Read: Motor standstill current, 16#6075 (Ch A)/ 16#6875 (Ch B)
		// Execute read only if DriveRef is OK
		IF bDriveRefOK THEN
			fbCoERead.nIndex			:= 16#6075 + 16#800 * stDriveRef.nDriveNo;
			fbCoERead.nSubIndex			:= 0;
			fbCoERead.pDstBuf			:= ADR(udiMotorStandstillCurrent);
			fbCoERead.cbBufLen			:= SIZEOF(udiMotorStandstillCurrent);
			fbCoERead.bExecute			:= TRUE;
			iStep 						:= iStep + 10; 
		END_IF
	
	10: // Wait till read finish
		IF NOT fbCoERead.bBusy THEN
			IF fbCoERead.bError THEN
				fbCoERead.bExecute		:= FALSE;
				wInitErrorCount 		:= wInitErrorCount + 1;
				// Count > 10 then go to error and wait for reset, if not wait in warning step
				IF wInitErrorCount > 10 THEN
					uiAdsErrId			:= fbCoERead.iAdsErrId;
					uiCANopenErrId		:= fbCoERead.iCANopenErrId;
					iStep				:= 1000;									// Error step
				ELSE
					iStep				:= 900;										// Warning step
				END_IF
			ELSE
				fbCoERead.bExecute		:= FALSE;
				iStep 					:= iStep + 10;
			END_IF
		END_IF
	
	20: // Read: Motor standstill torque 16#6076 (Ch A)/ 16#6876 (Ch B)
		// Execute read only if DriveRef is OK
		IF bDriveRefOK THEN
			fbCoERead.nIndex			:= 16#6076 + 16#800 * stDriveRef.nDriveNo;
			fbCoERead.nSubIndex			:= 0;
			fbCoERead.pDstBuf			:= ADR(udiMotorStandstillTorque);
			fbCoERead.cbBufLen			:= SIZEOF(udiMotorStandstillTorque);
			fbCoERead.bExecute			:= TRUE;
			iStep 						:= iStep + 10; 
		END_IF
	
	30:	// Wait till read finish
		IF NOT fbCoERead.bBusy THEN
			IF fbCoERead.bError THEN
				fbCoERead.bExecute		:= FALSE;
				wInitErrorCount 		:= wInitErrorCount + 1;
				// Count > 10 then go to error and wait for reset, if not wait in warning step
				IF wInitErrorCount > 10 THEN
					uiAdsErrId			:= fbCoERead.iAdsErrId;
					uiCANopenErrId		:= fbCoERead.iCANopenErrId;
					iStep				:= 1000;									// Error step
				ELSE
					iStep				:= 900;										// Warning step
				END_IF
			ELSE
				fbCoERead.bExecute		:= FALSE;
				iStep 					:= iStep + 10;
			END_IF
		END_IF
	
	40: // Calculate Sf
		rSfTorque						:= UDINT_TO_REAL(udiMotorStandstillTorque) / 1000000;
		rSfCurrent						:= UDINT_TO_REAL(udiMotorStandstillCurrent) / 1000000;
		rWarningCurrent					:= UDINT_TO_REAL(udiMotorStandstillCurrent) / 1000;
		iStep 							:= 100;
	
	100: // Read: Thermal Motor Utilization (I2T), 16#32C1:02 (Ch A)/ 16#36C1:02 (Ch B)
		fbCoERead.nIndex				:= 16#32C1 + (16#400 * stDriveRef.nDriveNo);
		fbCoERead.nSubIndex				:= 02;
		fbCoERead.pDstBuf				:= ADR(rI2T);
		fbCoERead.cbBufLen				:= SIZEOF(rI2T);
		fbCoERead.bExecute				:= bDriveRefOK AND tonWait.Q;				// Execute read only if DriveRef is OK
		IF fbCoERead.bBusy THEN
			iStep 						:= iStep + 10;
		END_IF
	
	110: // Wait till read finish
		IF NOT fbCoERead.bBusy THEN
			IF fbCoERead.bError OR NOT bTorqueLimitOK OR NOT bDriveRefOK THEN
				uiAdsErrId				:= fbCoERead.iAdsErrId;
				uiCANopenErrId			:= fbCoERead.iCANopenErrId;
				iStep					:= 1000;									// Error step
			ELSE
				iStep 					:= iStep - 10;				
			END_IF
		END_IF
	
	900: // Warning - wait and repeat read - problem during read motor data, i.e. EtherCAT doesn't work yet
		IF tonWait.Q THEN
			iStep 						:= 0;	// Repeat initialization phase 
		END_IF
			  
			  
	1000: // Error - wait for reset 
		;
END_CASE
//===============================================================
	 
bError			 						:= iStep = 1000;
bInitialized	 						:= iStep >= 100 AND NOT bError;
//====================== Call CoE read FB =======================
fbCoERead(stDriveRef:= stDriveRef);
//======================== Set outputs ==========================
rTorquePerc								:= LREAL_TO_REAL(Axis.NcToPlc.ActTorque); 		// [%]
rTorqueRAW 								:= rTorquePerc*10;								// -1000 .. 1000 - RAW values the same as process image
//===================== Filter current value ====================
fbFilterEx(rIn:= rTorqueRAW, tTimeConstant:= T#1S);

iTorque 								:= REAL_TO_INT(rTorqueRAW);
rTorque 								:= rTorqueRAW * rSfTorque;
rCurrent 								:= rTorqueRAW * rSfCurrent;
rTorqueF 								:= fbFilterEx.rOut * rSfTorque;
rCurrentF 								:= fbFilterEx.rOut * rSfCurrent;
//=============== Save torque and current max values ===============
IF ABS(rCurrentMax) < ABS(rCurrentF) THEN
	rTorquePercMax						:= rTorquePerc;
	rCurrentMax 						:= rCurrentF;
	rTorqueMax 							:= rTorqueF;
END_IF
//======================== Save I2T max value ======================
IF rI2TMax < rI2T THEN
	rI2TMax 							:= rI2T;
END_IF

//===================== Limit output torque =====================
IF rTorqueLimit < rTorqueLimitLow THEN
	uiBipolarTorqueLimitValue 			:= REAL_TO_UINT(rTorqueLimitHigh);			// Secure against 0 value - probably empty var connected to input
ELSE
	uiBipolarTorqueLimitValue 			:= REAL_TO_UINT(LIMIT(rTorqueLimitLow,rTorqueLimit,rTorqueLimitHigh))*10;
END_IF
//========================= Warning =============================
bWarning								:= rCurrentF > rWarningCurrent;

END_FUNCTION_BLOCK

// ---- POUs/POUsAxisOnline/AX8000/FB_ReadChannelErrorCodeAX8000.TcPOU
//==================================================================================================
//							Beckhoff Automation Poland
//									11.04.2018
//	This object shall provide the text id of the last DiagMessage of type error, which occurred in this axis.
//  v1.0	|| TC v 3.1.4022.16		|| - pierwsza wersja
//==================================================================================================
FUNCTION_BLOCK FB_ReadChannelErrorCodeAX8000
VAR_INPUT
	bExecute 						: BOOL;
	stDriveRef						: ST_DriveRef;						// 
END_VAR
VAR_OUTPUT
	bBusy							: BOOL;
	bError							: BOOL; 							// General error: parameter or CoE read.
	iAdsErrId						: UINT;								// Forwarded output FB_CoERead_ByDriveRef
	iCANopenErrId					: UINT;								// Forwarded output FB_CoERead_ByDriveRef
	uiChannelErrorCode				: UINT;								// 603F Error code	0x603F (Ch A)/ 0x683F (Ch B) 	UINT16
	{attribute 'displaymode':='hex'}
	uiChannelErrorCodeHex			: UINT;								// 603F Error code	0x603F (Ch A)/ 0x683F (Ch B) 	UINT16
END_VAR
VAR
	fbCoERead						: FB_CoERead_ByDriveRef;			// FB for read CoE parameters
END_VAR

fbCoERead(	stDriveRef					:= stDriveRef,
			nIndex						:= 16#603F + (stDriveRef.nDriveNo * 16#800),
			nSubIndex					:= 0,
			pDstBuf						:= ADR(uiChannelErrorCode),
			cbBufLen					:= SIZEOF(uiChannelErrorCode),
			bExecute					:= bExecute,
			bBusy						=> bBusy,
			bError						=> bError,
			iAdsErrId					=> iAdsErrId,
			iCANopenErrId				=> iCANopenErrId);

uiChannelErrorCodeHex					:= uiChannelErrorCode;

END_FUNCTION_BLOCK

// ---- POUs/POUsAxisOnline/AX8000/F_AX8xErrMsg.TcPOU
//==================================================================================================
//							Beckhoff Automation Poland
//								7.12.2018
//		Funkcja konwertujaca nr bledu na opis
// 	v1.0	|| TC v 3.1.4022.27	|| - pierwsza wersja
//==================================================================================================
FUNCTION F_AX8xErrMsg : STRING(255)
VAR_INPUT
	uiDriveError : UINT;
END_VAR

IF uiDriveError < 1 THEN
	F_AX8xErrMsg := '';
	RETURN;
END_IF

CASE uiDriveError OF
	16#2220: F_AX8xErrMsg:= '2220 =  Continuous over current (device internal)';
	16#2310: F_AX8xErrMsg:= '2310 =  Continuous over current (device output side)';
	16#2330: F_AX8xErrMsg:= '2330 = Earth leakage (motor-side)';
	16#2340: F_AX8xErrMsg:= '2340 =  Short circuit (motor-side)';
	16#2380: F_AX8xErrMsg:= '2380 =  Continuous over current (device output side) Phase U';
	16#2381: F_AX8xErrMsg:= '2381 =  Continuous over current (device output side) Phase V';
	16#2382: F_AX8xErrMsg:= '2382 =  Continuous over current (device output side) Phase W';
	16#2383: F_AX8xErrMsg:= '2383 =  Phase U current offset out of range';
	16#2384: F_AX8xErrMsg:= '2384 =  Phase V current offset out of range';
	16#2385: F_AX8xErrMsg:= '2385 =  Phase W current offset out of range';
	16#3110: F_AX8xErrMsg:= '3110 =  Mains over-voltage';
	16#3120: F_AX8xErrMsg:= '3120 =  Mains under-voltage';
	16#3130: F_AX8xErrMsg:= '3130 =  Phase failure';
	16#3180: F_AX8xErrMsg:= '3180 =  Phase failure motor or Mains voltage over brake resistor operating voltage';
	16#3181: F_AX8xErrMsg:= '3181 =  Phase frequency (motor-side) raised above 600 Hz or Wrong mains type';
	16#3182: F_AX8xErrMsg:= '3182 =  Velocity actual Value raised above the max channel accepted velocity';
	16#3183: F_AX8xErrMsg:= '3183 = The bipolar velocity limit is higher than 1/4 of position range limit per EtherCAT Sync1 cycle.';
	16#3210: F_AX8xErrMsg:= '3210 =  DC link over-voltage';
	16#3220: F_AX8xErrMsg:= '3220 =  DC link undervoltage';
	16#3280: F_AX8xErrMsg:= '3280 =  DC link is not ready or  Device DC link over-voltage';
	16#4110: F_AX8xErrMsg:= '4110 =  Excess ambient temperature';
	16#4210: F_AX8xErrMsg:= '4210 =  Excess temperature device';
	16#4310: F_AX8xErrMsg:= '4310 =  Drive overtemperature shut down';
	16#4380: F_AX8xErrMsg:= '4380 =  Fan speed seems to be zero.';
	16#5112: F_AX8xErrMsg:= '5112 =  Supply low voltage: supply +24V';
	16#5180: F_AX8xErrMsg:= '5180 =  Output stage STO active.';
	16#5181: F_AX8xErrMsg:= '5181 =  Power supply status,  torque off order';
	16#5182: F_AX8xErrMsg:= '5182 =  Power supply status inactive';
	16#5183: F_AX8xErrMsg:= '5183 =  Power supply status,  NC handling order';
	16#5184: F_AX8xErrMsg:= '5184 =  Supply DC-link circuit is not ready';
	16#5185: F_AX8xErrMsg:= '5185 =  Power supply status,  non-regenerative brake order';
	16#5186: F_AX8xErrMsg:= '5186 =  Power supply status,  regenerative brake order';
	16#5187: F_AX8xErrMsg:= '5187 =  Power supply communication is not established';
	16#5190: F_AX8xErrMsg:= '5190 =  Test 5V supply failed';
	16#5192: F_AX8xErrMsg:= '5192 =  Supply high voltage: supply +24V';
	16#5441: F_AX8xErrMsg:= '5441 =  Positive limit switch active';
	16#5442: F_AX8xErrMsg:= '5442 =  Negative limit switch active';
	16#5580: F_AX8xErrMsg:= '5580 =  Read failure EEPROM';
	16#5581: F_AX8xErrMsg:= '5581 =  Checksum failure EEPROM';
	16#5582: F_AX8xErrMsg:= '5582 =  EEPROM contains blank Data';
	16#5583: F_AX8xErrMsg:= '5583 =  Unexpected EEPROM';
	16#5584: F_AX8xErrMsg:= '5584 =  EEPROM contains blank Data';
	16#5585: F_AX8xErrMsg:= '5585 =  Unexpected EEPROM';
	16#5586: F_AX8xErrMsg:= '5586 =  Restored Errormessages from persistant memory';
	16#5587: F_AX8xErrMsg:= '5587 =  Missing factory settings in eeprom';
	16#5588: F_AX8xErrMsg:= '5588 =  Missing ids in eeprom display board';
	16#5589: F_AX8xErrMsg:= '5589 =  Read failure eeprom display board';
	16#5590: F_AX8xErrMsg:= '5590 =  Detected incompatible Pcb';
	16#5591: F_AX8xErrMsg:= '5591 =  Identity incompatible to a Pcb';
	16#5592: F_AX8xErrMsg:= '5592 =  FirmwareIndex is incompatible to this Firmware.';
	16#5593: F_AX8xErrMsg:= '5593 =  Structure Version is incompatible to this Firmware';
	16#5594: F_AX8xErrMsg:= '5594 =  Simulating persistent data features.';
	16#5595: F_AX8xErrMsg:= '5595 =  Modulo remainder will not be stored.';
	16#5596: F_AX8xErrMsg:= '5596 =  Storing of persistant data failed.';
	16#6010: F_AX8xErrMsg:= '6010 =  Software reset (watchdog)';
	16#6080: F_AX8xErrMsg:= '6080 =  Failure config bits';
	16#6180: F_AX8xErrMsg:= '6180 =  Internal Software Error Type A';
	16#6181: F_AX8xErrMsg:= '6181 =  Internal Software Error Type B';
	16#6182: F_AX8xErrMsg:= '6182 =  Internal Software Error Type C';
	16#6183: F_AX8xErrMsg:= '6183 =  Internal Watchdog Error';
	16#6190: F_AX8xErrMsg:= '6190 =  Init Timeout';
	16#6310: F_AX8xErrMsg:= '6310 =  Loss of parameters';
	16#6320: F_AX8xErrMsg:= '6320 =  Parameter error';
	16#6380: F_AX8xErrMsg:= '6380 =  Parameter Interpolator: Illegal Interpolation sub mode select or  Parameters x with parametrized y is too low.';
	16#6381: F_AX8xErrMsg:= '6381 =  Parameter x with parametrized y is too high';
	16#6382: F_AX8xErrMsg:= '6382 =  Illegal Slotconfiguration. Slot is empty.';
	16#6383: F_AX8xErrMsg:= '6383 =  Illegal Slotconfiguration. Double Feedback Selection.';
	16#6384: F_AX8xErrMsg:= '6384 =  Illegal Slotconfiguration. Slot has to be empty.';
	16#6385: F_AX8xErrMsg:= '6385 =  Parameter Interpolator. Operation Mode does not match';
	16#6386: F_AX8xErrMsg:= '6386 =  Parameter Interpolator: Illegal NC-Task cycle time';
	16#6387: F_AX8xErrMsg:= '6387 =  Parameter Motor. The configured DCLink Max Voltage is higher than the Motor Max Voltage.';
	16#6388: F_AX8xErrMsg:= '6388 =  Parameter Torque Control: The value in Object 0x%x/%x is higher than the Motor peak current (0x%x/%x).';
	16#6389: F_AX8xErrMsg:= '6389 =  Parameter Torque Control: The value in Object 0x%x/%x is higher than the Configured peak current (0x%x/%x).';
	16#6390: F_AX8xErrMsg:= '6390 =  Factor Group Parameters: Feed constant illegal feed';
	16#6391: F_AX8xErrMsg:= '6391 =  Factor Group Parameters: Feed constant illegal shaft revolutions';
	16#6392: F_AX8xErrMsg:= '6392 =  Factor Group Parameters: Gear ratio illegal Motor shaft revolutions';
	16#6393: F_AX8xErrMsg:= '6393 =  Factor Group Parameters: Gear ratio illegal Driving shaft revolutions';
	16#6394: F_AX8xErrMsg:= '6394 =  Factor Group Parameters: Position encoder resolution illegal encoder increments';
	16#6395: F_AX8xErrMsg:= '6395 =  Factor Group Parameters: Position encoder resolution illegal motor revolutions';
	16#6396: F_AX8xErrMsg:= '6396 =  additional Factor Group Parameters: Feed constant illegal feed';
	16#6397: F_AX8xErrMsg:= '6397 =  additional Factor Group Parameters: Feed constant illegal shaft revolutions';
	16#6398: F_AX8xErrMsg:= '6398 =  additional Factor Group Parameters: Gear ratio illegal Motor shaft revolutions';
	16#6399: F_AX8xErrMsg:= '6399 =  additional Factor Group Parameters: Gear ratio illegal Driving shaft revolutions';
	16#7111: F_AX8xErrMsg:= '7111 =  Failure brake chopper';
	16#7112: F_AX8xErrMsg:= '7112 =  Over current brake chopper';
	16#7122: F_AX8xErrMsg:= '7122 =  Motor error or commutation malfunction';
	16#7180: F_AX8xErrMsg:= '7180 =  Motor brake: Current monitoring error. Or  Brake resistor not found';
	16#7181: F_AX8xErrMsg:= '7181 =  Motor thermal utilization has reached the warning level.  Or  Brake resistor power overload by DC link over-voltage';
	16#7182: F_AX8xErrMsg:= '7182 =  Motor thermal utilization has left the warning level. Or  Wrong xml file';
	16#7183: F_AX8xErrMsg:= '7183 =  Motor thermal utilization has reached the Error Level';
	16#7184: F_AX8xErrMsg:= '7184 =  Motor overload shut down';
	16#7185: F_AX8xErrMsg:= '7185 =  Motor overtemperature shut down';
	16#7186: F_AX8xErrMsg:= '7186 = Detected moving axis on enable transition.';
	16#7320: F_AX8xErrMsg:= '7320 =  HpfDsl: Encoder error (position invalid)';
	16#7380: F_AX8xErrMsg:= '7380 =  Current sensor motor phase U or HpfDsl: Encoder start sequence failed';
	16#7381: F_AX8xErrMsg:= '7381 =  Current sensor motor phase V or HpfDsl: Encoder shutdown failed';
	16#7382: F_AX8xErrMsg:= '7382 =  Current sensor motor phase W or HpfDsl: Parameter access error';
	16#7383: F_AX8xErrMsg:= '7383 =  HpfDsl: Internal error';
	16#7384: F_AX8xErrMsg:= '7384 =  HpfDsl: Cyclic monitoring error';
	16#7385: F_AX8xErrMsg:= '7385 =  HpfDsl: Encoder file processing';
	16#7386: F_AX8xErrMsg:= '7386 =  HpfDsl: Found no encoder (No link to an encoder)!';
	16#7580: F_AX8xErrMsg:= '7580 =  I2C_communication_failure';
	16#8180: F_AX8xErrMsg:= '8180 =  System restart or sync lost';
	16#8181: F_AX8xErrMsg:= '8181 =  Lost Distributed clocks Sync';
	16#8182: F_AX8xErrMsg:= '8182 =  EtherCAT Statemachine shutdown with enabled Axis';
	16#8183: F_AX8xErrMsg:= '8183 =  Controlword output cycle counter monitoring';
	16#8480: F_AX8xErrMsg:= '8480 = Overspeed error';
	16#8611: F_AX8xErrMsg:= '8611 = Following error';
	16#8680: F_AX8xErrMsg:= '8680 =  Position Demand Value outside of the specified Position Range Limits';
	16#8780: F_AX8xErrMsg:= '8780 =  Configured Sync1 Cycle Time is above Maximum';
	16#8781: F_AX8xErrMsg:= '8781 =  Configured Sync1 Cycle Time is below Minimum';
	16#8782: F_AX8xErrMsg:= '8782 =  Configured Sync1 Cycle Time is not a multiple of the Sync0 Cycle Time';
	16#8783: F_AX8xErrMsg:= '8783 =  Configured Sync0 Cycle Time is not legal';
	16#638A: F_AX8xErrMsg:= '638A =  The Axis seems not to be parameterised.';
	16#638B: F_AX8xErrMsg:= '638B =  Parameter Torque Current curve: Unable to calculate Torque Current curve.';
	16#638C: F_AX8xErrMsg:= '638C =  Motor type does not match';
	16#638D: F_AX8xErrMsg:= '638D =  Connected Motor is compatible to the configured Motor';
	16#638E: F_AX8xErrMsg:= '638E =  The Motor brake is automatically unlocked';
	16#638F: F_AX8xErrMsg:= '638F =  Parameter Torque Control: The value in Object 0x%x/%x is higher then the Motor maximum voltage slope (0x%x/%x).';
	16#639A: F_AX8xErrMsg:= '639A =  additional Factor Group Parameters: Position encoder resolution illegal encoder increments';
	16#639B: F_AX8xErrMsg:= '639B =  additional Factor Group Parameters: Position encoder resolution illegal motor revolutions';
	16#639C: F_AX8xErrMsg:= '639C =  Velocity factor illegal. A possible Value would be %u/%u.';
	16#639D: F_AX8xErrMsg:= '639D =  Acceleration factor illegal. A possible Value would be %u/%u.';
	16#639E: F_AX8xErrMsg:= '639E =  Scaling index object 0x%x does not fit the Factor group parameters for the first Encoder';
	16#639F: F_AX8xErrMsg:= '639F =  Scaling index object 0x%x does not fit the Factor group parameters for the second Encoder';
	16#63A0: F_AX8xErrMsg:= '63A0 =  Motor or Primary Feedback changed';
	16#63A1: F_AX8xErrMsg:= '63A1 =  Secondary Feedback changed';
	16#63A2: F_AX8xErrMsg:= '63A2 =  Offset position actual value: No position offset existing in source "encoder memory"';
	16#63A3: F_AX8xErrMsg:= '63A3 =  Offset additional position actual value: No position offset existing in source "encoder memory"';
	16#63A4: F_AX8xErrMsg:= '63A4 =  Offset position actual value: No position offset existing in source "drive memory"';
	16#63A5: F_AX8xErrMsg:= '63A5 =  Offset additional position actual value: No position offset existing in source "drive memory"';
	16#63A6: F_AX8xErrMsg:= '63A6 =  Jerk factor illegal. A possible Value would be %u/%u.';
	16#63A7: F_AX8xErrMsg:= '63A7 =  The range %u of the Position range limit is below the minimum accepted value of %u.';
	16#63A8: F_AX8xErrMsg:= '63A8 =  Position range limit Inc with remainder is not supported for primary feedback.';
	16#63A9: F_AX8xErrMsg:= '63A9 =  Position range limit Inc with remainder is not supported for secondary feedback.';
	16#63AA: F_AX8xErrMsg:= '63AA =  Object 0x%X/%X changed in EtherCAT SafeOP or OP.';
	16#8A80: F_AX8xErrMsg:= '8A80 =  Illegal Modes of Operation';
	16#8A81: F_AX8xErrMsg:= '8A81 =  Illegal Modes of Operation change';
	16#A000: F_AX8xErrMsg:= 'A000 =  Transition Pre-Op to Safe-Op not successful. Sync Manager Length Error.';
	16#A001: F_AX8xErrMsg:= 'A001 =  Transition Pre-Op to Safe-Op not successful. Sync Manager Address Error.';
	16#A002: F_AX8xErrMsg:= 'A002 =  Transition Pre-Op to Safe-Op not successful. Sync Manager Settings Error.';
	16#A003: F_AX8xErrMsg:= 'A003 =  Transition Pre-Op to Safe-Op not successful. Sync Manager Address Range overlap.';
	16#A004: F_AX8xErrMsg:= 'A004 =  Sync Manager is disabledand has a Size unequal zero.';
	16#A010: F_AX8xErrMsg:= 'A010 =  SDO Complete Access Error: Object 0x%x/%x';
	16#A011: F_AX8xErrMsg:= 'A011 =  RxPdo Mapping Error: Unable to map Object (not possible).';
	16#A012: F_AX8xErrMsg:= 'A012 =  TxPdo Mapping Error: Unable to map Object (not possible).';
	16#A013: F_AX8xErrMsg:= 'A013 =  RxPdo Mapping Error: Double Mapping of Object.';
	16#A014: F_AX8xErrMsg:= 'A014 =  TxPdo Mapping Error: Double Mapping of Object.';
	16#A015: F_AX8xErrMsg:= 'A015 =  RxPdo Mapping Error: Unable to map Object (no Mappings left).';
	16#A016: F_AX8xErrMsg:= 'A016 =  TxPdo Mapping Error: Unable to map Object (no Mappings left).';
	16#A017: F_AX8xErrMsg:= 'A017 =  RxPdo Mapping Error: Object always has to be mapped.';
	16#A018: F_AX8xErrMsg:= 'A018 =  TxPdo Mapping Error: Object 0x%x/%x always has to be mapped.';
	16#A019: F_AX8xErrMsg:= 'A019 =  RxPdo Mapping Error: Object has to be mapped because of modes of operation.';
	16#A01A: F_AX8xErrMsg:= 'A01A =  TxPdo Mapping Error: Object has to be mapped because of modes of operation.';
	16#A01B: F_AX8xErrMsg:= 'A01B =  RxPdo BitMapping Error: Object 0x%x/%x is not next to Object 0x%x/%x. (SyncManager %u)';
	16#A01C: F_AX8xErrMsg:= 'A01C =  TxPdo BitMapping Error: Object 0x%x/%x is not next to Object 0x%x/%x. (SyncManager %u)';
	16#A01D: F_AX8xErrMsg:= 'A01D =  RxPdo BitMapping Error: Can not Transform Bit-Mappings to Byte-Mappings. (SyncManager %u)';
	16#A01E: F_AX8xErrMsg:= 'A01E =  TxPdo BitMapping Error: Can not Transform Bit-Mappings to Byte-Mappings. (SyncManager %u)';
	16#A080: F_AX8xErrMsg:= 'A080 =  Safe-Op is not possible because the local TwinCAT Runtime is in ConfigMode.';
	16#A081: F_AX8xErrMsg:= 'A081 =  Transition Pre-Op to Safe-Op not successful. Safetycard not detected.';
	16#A082: F_AX8xErrMsg:= 'A082 =  EtherCAT Slave Stack Error:';
	16#FF01: F_AX8xErrMsg:= 'FF01 =  Init Timeout or Error reaction forced: Generative brake order';
	16#FF02: F_AX8xErrMsg:= 'FF02 =  Error reaction forced: Non-generative brake order';
	16#FF03: F_AX8xErrMsg:= 'FF03 =  Error reaction forced: Brake chopper off';
	16#FF07: F_AX8xErrMsg:= 'FF07 =  Error reaction forced: Torque Off';
	16#FF08: F_AX8xErrMsg:= 'FF08 =  Error reaction forced: Shorted Coils Brake';
	16#FF09: F_AX8xErrMsg:= 'FF09 =  Error reaction forced: Open Loop Ramp';
	16#FF0A: F_AX8xErrMsg:= 'FF0A =  Error reaction forced: Closed Loop Ramp';
	16#FF0B: F_AX8xErrMsg:= 'FF0B =  Error reaction forced: NC handling';
	16#FF0C: F_AX8xErrMsg:= 'FF0C =  Error reaction TorqueOff with emergency brake';
	16#FFFC: F_AX8xErrMsg:= 'FFFC =  %s';
	16#FFFD: F_AX8xErrMsg:= 'FFFD =  Debug firmware.  Replace "As soon as possible"!';
	16#FFFE: F_AX8xErrMsg:= 'FFFE =  %s';
	16#FFFF: F_AX8xErrMsg:= 'FFFF =  Internal Error.   Additional Errorcode 0x%x';

ELSE
	F_AX8xErrMsg := UINT_TO_STRING(uiDriveError);
	F_AX8xErrMsg := concat(F_AX8xErrMsg, ' Unknown Error code');
END_CASE
F_AX8xErrMsg := F_AX8xErrMsg;

END_FUNCTION

// ---- POUs/POUsAxisOnline/EL72xx/FB_HoldingBrakeCtrlEL72xx.TcPOU
//==================================================================================================
//							Beckhoff Automation Poland
//									11.07.2018
//	Blok funkcyjny kontroli luzownika w silniku podpietym do EL72xx. Mozliwy jest jedynie force unlock.
//	Dzialania na obiekcie:	: 8012:01 (MDP742) lub 2004:01 (DS402)
//
//  v1.0	|| TC v 3.1.4022.22		|| - pierwsza wersja
//==================================================================================================
FUNCTION_BLOCK FB_HoldingBrakeCtrlEL72xx
VAR_INPUT
	bForceUnlock					: BOOL;								// Rising/falling edhe executes CMD: Manual override (release) of the motor holding brake 
																		// and reset - if there is error - falling edge reinits FB
	stDriveRef						: ST_DriveRef;
END_VAR
VAR_OUTPUT
	bBusy							: BOOL;
	bError							: BOOL; 							// General error: parameter or CoE read.
	uiAdsErrId						: UINT;								// Forwarded output FB_CoERead_ByDriveRef
	uiCANopenErrId					: UINT;								// Forwarded output FB_CoERead_ByDriveRef
END_VAR
VAR
	//======================= Internal var ===========================
	iStep							: INT;								// Case instruction	
	wInitErrorCount					: WORD;								// Initialization error counter, if bigger then 10 then error
	wManualOverrideIndex			: WORD;								// Manual override (release) of the motor holding brake:
																		// MDP742: 8012:01
																		// DS402: 2004:01
	bDriveRefOK						: BOOL;								// stDriveRef contains necessary data to read CoE
	bExecute						: BOOL;
	bDS402Profile					: BOOL;								// Flag DS402
	bMDP742Profile					: BOOL;								// Flag MDP742	
	bInitialized					: BOOL;
	sDeviceName						: STRING;							// 
	sNo								: STRING(1);						// xxxxxxx-000Y - char Y	
	//=========================== FBs ================================																
	rtForceUnlock					: R_TRIG;
	ftForceUnlock					: F_TRIG;
	tonWait							: TON;								// Wait timer
	fbCoERead						: FB_CoERead_ByDriveRef;			// FB for read CoE parameters
	fbForceUnlock					: FB_CoEWrite_ByDriveRef;
END_VAR

//=================== Call triggers and timers ==================
tonWait(IN:= NOT tonWait.Q, PT:= T#1S);
rtForceUnlock(CLK:= bForceUnlock);
ftForceUnlock(CLK:= bForceUnlock);

//======= Check for parameter error - each cycle ================
bDriveRefOK 							:= (stDriveRef.nSlaveAddr <> 0) AND (stDriveRef.sNetId <> '');

//============= Read params and calculations ====================
CASE iStep OF
	
	0: // Read profile MDP 742 or DS 402:
	
			// We have to read device name Index 1008:0 - STRING
			// EL72x1-0000 --> MDP 742:
			// EL72x1-0001 --> DS 402:
	
		// Execute read only if DriveRef is OK
		IF bDriveRefOK THEN
			fbCoERead.nIndex			:= 16#1008;
			fbCoERead.nSubIndex			:= 0;
			fbCoERead.pDstBuf			:= ADR(sDeviceName);
			fbCoERead.cbBufLen			:= SIZEOF(sDeviceName);
			fbCoERead.bExecute			:= TRUE;
			iStep 						:= iStep + 10; 
		END_IF
	
	10:	// Wait till read finish
	
		IF NOT fbCoERead.bBusy THEN
			fbCoERead.bExecute			:= FALSE;
			IF fbCoERead.bError THEN
				wInitErrorCount 		:= wInitErrorCount + 1;
				// Count > 10 then go to error and wait for reset, if not wait in warning step
				IF wInitErrorCount > 10 THEN
					uiAdsErrId			:= fbCoERead.iAdsErrId;
					uiCANopenErrId		:= fbCoERead.iCANopenErrId;
					iStep				:= 1000;								// Error step
				ELSE
					iStep				:= 900;									// Warning step
				END_IF
			ELSE
				iStep 					:= iStep + 10;
			END_IF
		END_IF

	20: // Check last digit in device name 0 - MDP742, 1 - DS402
	
	sNo 								:=  MID(sDeviceName, 1, FIND(sDeviceName, '-') + 4);
	bMDP742Profile 						:= 	sNo = '0';
	bDS402Profile 						:= 	sNo = '1';
	// If 0 or 1 then go to next step, if other No - not implemented yet
	IF bMDP742Profile OR bDS402Profile THEN
		wManualOverrideIndex			:= SEL(bMDP742Profile, 16#2004, 16#8012);
		iStep 							:= 100;
	ELSE
		iStep							:= 1000;					// Error step
	END_IF
	
	100: // Initialized - holding brake control possible
		fbForceUnlock.bExecute			:= rtForceUnlock.Q OR ftForceUnlock.Q;
		IF fbForceUnlock.bBusy THEN
			iStep 						:= iStep + 10;
		END_IF

	110: // Wait till write finish
	
		IF NOT fbForceUnlock.bBusy THEN
			fbForceUnlock.bExecute		:= FALSE;
			IF fbForceUnlock.bError THEN
				uiAdsErrId				:= fbForceUnlock.iAdsErrId;
				uiCANopenErrId			:= fbForceUnlock.iCANopenErrId;
			ELSE
				iStep 					:= iStep - 10;
			END_IF
		END_IF
	
	900: // Warning - wait and repeat read - problem during read motor data, i.e. EtherCAT doesn't work yet
		IF tonWait.Q THEN
			iStep 						:= 0;	// Repeat initialization phase 
		END_IF
			  
	1000: // Error - wait for reset 
		IF ftForceUnlock.Q THEN
			uiAdsErrId					:= 0;
			uiCANopenErrId				:= 0;
			wInitErrorCount				:= 0;
			wManualOverrideIndex		:= 0;
			sDeviceName					:= '';
			sNo							:= '';
			bDS402Profile				:= FALSE;
			bMDP742Profile				:= FALSE;
			iStep						:= 0;
		END_IF
END_CASE
//===============================================================

bError		 							:= iStep = 1000;
bInitialized 							:= iStep >= 100 AND iStep < 900;

//================== Call CoE read/write FB =====================
fbCoERead(stDriveRef:= stDriveRef);

fbForceUnlock	(	stDriveRef				:= stDriveRef, 
					nIndex					:= wManualOverrideIndex, 
					nSubIndex				:= 16#01, 
					pSrcBuf					:= ADR(bForceUnlock), 
					cbBufLen				:= SIZEOF(bForceUnlock));
//===============================================================

END_FUNCTION_BLOCK

// ---- POUs/POUsAxisOnline/EL72xx/FB_McAxisOnlineEL72xx.TcPOU
//==================================================================================================
//							Beckhoff Automation Poland
//									7.12.2018
//	Wszystkomajacy blok funkcyjny do sterowania osia, 
//	wymagane biblioteki: Tc2_EtherCAT, Tc2_MC2_Drive, Tc2_MC2
//  v1.1	|| TC v 3.1.4022.27		|| - dodane opisy bledow w formie zmiennych typu string
// 	v1.0 	|| TC v 3.1.4022.22	 	|| - first edition
//==================================================================================================
{attribute 'reflection'}
FUNCTION_BLOCK FB_McAxisOnlineEL72xx
VAR_IN_OUT
	stMcAxisOnline						: ST_McAxisOnline;
	Axis								: AXIS_REF;
END_VAR
VAR
	mcPower								: MC_Power;
	mcStop								: MC_Stop;
	mcHalt								: MC_Halt;
	mcStopSS1							: MC_Stop;
	mcStopSS2							: MC_Stop;
	mcReset								: MC_Reset;
	mcHome								: MC_Home;
	mcSetPosition						: MC_SetPosition;
	fbSetPositionOffset					: FB_CoEEL72xxSetPositionOffset;// Not Yet avaliable
	mcJog								: MC_Jog;

	mcMoveAbsolute						: MC_MoveAbsolute;
	mcMoveRelative						: MC_MoveRelative;
	mcMoveVelocity						: MC_MoveVelocity;
	mcMoveModulo						: MC_MoveModulo;
	mcMoveAbsolute2						: MC_MoveAbsolute;
	mcMoveRelative2						: MC_MoveRelative;
	mcMoveVelocity2						: MC_MoveVelocity;
	mcMoveModulo2						: MC_MoveModulo;

	fbMotorMonitoring					: FB_MotorMonitoringEL72xx;
	fbHoldingBrakeCtrl					: FB_HoldingBrakeCtrlEL72xx;
	fbNcLimitSwitch						: FB_NcSWLimitSwitchCtrl;
	tonGetDriveDiag						: TON;
	fbReadChannelErrorCode				: FB_ReadChannelErrorCodeEL72xx;
	
	mcReadDriveAddress					: MC_ReadDriveAddress;
	mcReadParameterSet					: MC_ReadParameterSet;
	fbGetDriveRef						: FB_GetDriveRef;

	// Internal
	bInitialized						: BOOL;
	bCommError							: BOOL;
	bReadParameterError					: BOOL;
	bInitError							: BOOL;
	bDriveError							: BOOL;
	bFBError							: BOOL;
	
// Initialization
	iInitStep							: INT;
	bInitializationError				: BOOL;
	wInitializationErrorCounter			: WORD;
	bDriveAddressReady					: BOOL;
	bDriveRefReady						: BOOL;
	bReadParameterSetReady				: BOOL;
	tonDelay							: TON;
// Re init
	udiOnlineChangeCntOld				: UDINT;
	bOnlineChangeDetected				: BOOL;
	bReInit								: BOOL;
	bReInitialized						: BOOL;
	bReInitializationError				: BOOL;
	{attribute 'instance-path'}
	{attribute 'noinit'}
	sInstancePath						: STRING;
END_VAR

// Device dependent initialization 
ACT_Initialization();
// Device independent commands, mostly NC 
ACT_States();
ACT_SWLimitSwitch();
ACT_Stop();
ACT_Power();
ACT_Homing();
ACT_Jog();
ACT_Move();
ACT_Reset();
ACT_SetPosition();
// Device dependent commands
// Motor monitoring possible only with real axis
IF NOT Axis.Status.OpMode.SimulationAxis THEN
	ACT_MotorMonitoring();
END_IF
// Device dependent commands, possible only on real axis after complete initialization
IF bInitialized AND NOT Axis.Status.OpMode.SimulationAxis THEN
	ACT_SetPositionIO();
	ACT_DriveDiag();
	ACT_HoldingBrakeCtrl();
END_IF

// Device independent error collection
ACT_ErrorCollection();

ACTION ACT_DriveDiag:
// Auto update when drive error
tonGetDriveDiag(IN:= stMcAxisOnline.stError.bDriveError AND NOT tonGetDriveDiag.Q, PT:= T#5S, Q=> , ET=> );

fbReadChannelErrorCode(	bExecute				:= stMcAxisOnline.stChannelErrorCode.bExecute OR tonGetDriveDiag.Q,
						stDriveRef				:= stMcAxisOnline.stDriveRef,
						bBusy					=> stMcAxisOnline.stChannelErrorCode.bBusy,
						bError					=> stMcAxisOnline.stChannelErrorCode.bError,
						uiAdsErrId				=> stMcAxisOnline.stChannelErrorCode.uiAdsErrId,
						uiCANopenErrId			=> stMcAxisOnline.stChannelErrorCode.uiSecErrId,
						uiChannelErrorCode		=> stMcAxisOnline.stChannelErrorCode.uiChannelErrorCode,
						uiChannelErrorCodeHex	=> stMcAxisOnline.stChannelErrorCode.uiChannelErrorCodeHex);
END_ACTION

ACTION ACT_ErrorCollection:
// Error flags
stMcAxisOnline.stError.bDriveError					:= Axis.Status.DriveDeviceError;

stMcAxisOnline.stError.bNcError						:= Axis.Status.Error;

stMcAxisOnline.stError.bFBError						:= stMcAxisOnline.mcPower.bError OR stMcAxisOnline.mcReset.bError OR stMcAxisOnline.mcHome.bError OR stMcAxisOnline.mcJog.bError
													OR stMcAxisOnline.mcHalt.bError OR stMcAxisOnline.mcStop.bError OR stMcAxisOnline.mcSS1.bError OR stMcAxisOnline.mcSS2.bError
													OR stMcAxisOnline.mcMoveAbsolute.bError OR stMcAxisOnline.mcMoveRelative.bError OR stMcAxisOnline.mcMoveVelocity.bError OR stMcAxisOnline.mcMoveModulo.bError
													OR stMcAxisOnline.mcMoveAbsolute2.bError OR stMcAxisOnline.mcMoveRelative2.bError OR stMcAxisOnline.mcMoveVelocity2.bError OR stMcAxisOnline.mcMoveModulo2.bError
													OR stMcAxisOnline.stNcLimitSwitch.bError OR stMcAxisOnline.mcSetPosition.bError;
									
stMcAxisOnline.stError.bCommunicationError			:= stMcAxisOnline.stChannelErrorCode.bError OR stMcAxisOnline.stSetPositionOffset.bError OR stMcAxisOnline.stMotorMonitoring.bError OR stMcAxisOnline.stHoldingBrake.bError;

stMcAxisOnline.stError.bError						:= stMcAxisOnline.stError.bDriveError OR stMcAxisOnline.stError.bNcError OR stMcAxisOnline.stError.bFBError OR stMcAxisOnline.stError.bCommunicationError;
stMcAxisOnline.bError								:= stMcAxisOnline.stError.bError; // Forward one stage up

// Error codes
stMcAxisOnline.stError.uiDriveErrorID 				:= stMcAxisOnline.stChannelErrorCode.uiChannelErrorCode;
stMcAxisOnline.stError.uiDriveErrorIDHex 			:= stMcAxisOnline.stChannelErrorCode.uiChannelErrorCodeHex;

stMcAxisOnline.stError.udiNcErrorID 				:= Axis.Status.ErrorID;
stMcAxisOnline.stError.udiNcErrorIDHex 				:= Axis.Status.ErrorID;
	

stMcAxisOnline.stError.udiFBErrorID 				:= 	stMcAxisOnline.mcPower.udiErrorID + 
														stMcAxisOnline.mcReset.udiErrorID + 
														stMcAxisOnline.mcHome.udiErrorID + 
														stMcAxisOnline.mcJog.udiErrorID +
														stMcAxisOnline.mcHalt.udiErrorID + 
														stMcAxisOnline.mcStop.udiErrorID + 
														stMcAxisOnline.mcSS1.udiErrorID + 
														stMcAxisOnline.mcSS2.udiErrorID +
														stMcAxisOnline.mcMoveAbsolute.udiErrorID + 
														stMcAxisOnline.mcMoveRelative.udiErrorID + 
														stMcAxisOnline.mcMoveVelocity.udiErrorID + 
														stMcAxisOnline.mcMoveModulo.udiErrorID +
														stMcAxisOnline.mcMoveAbsolute2.udiErrorID + 
														stMcAxisOnline.mcMoveRelative2.udiErrorID + 
														stMcAxisOnline.mcMoveVelocity2.udiErrorID + 
														stMcAxisOnline.mcMoveModulo2.udiErrorID +
														stMcAxisOnline.stNcLimitSwitch.udiErrorID + 
														stMcAxisOnline.mcSetPosition.udiErrorID;

stMcAxisOnline.stError.udiFBErrorIDHex 				:= stMcAxisOnline.stError.udiFBErrorID;

stMcAxisOnline.stError.udiErrorID					:= stMcAxisOnline.stSetPositionOffset.udiErrorID;
stMcAxisOnline.stError.uiAdsErrorID					:= stMcAxisOnline.stChannelErrorCode.uiAdsErrId + stMcAxisOnline.stMotorMonitoring.uiAdsErrId + stMcAxisOnline.stHoldingBrake.uiAdsErrId;
stMcAxisOnline.stError.uiSecErrorID					:= stMcAxisOnline.stChannelErrorCode.uiSecErrId + stMcAxisOnline.stMotorMonitoring.uiSecErrId + stMcAxisOnline.stHoldingBrake.uiSecErrId;

stMcAxisOnline.stError.sNcError						:= F_AxErrMsg(stMcAxisOnline.stError.udiNcErrorID);
stMcAxisOnline.stError.sDriveError					:= F_EL72ErrMsg(stMcAxisOnline.stError.uiDriveErrorID);
END_ACTION

ACTION ACT_HoldingBrakeCtrl:
fbHoldingBrakeCtrl(bForceUnlock		:= stMcAxisOnline.stHoldingBrake.bForceUnlock,
					stDriveRef			:= stMcAxisOnline.stDriveRef,
					bBusy				=> stMcAxisOnline.stHoldingBrake.bBusy,
					bError				=> stMcAxisOnline.stHoldingBrake.bError,
					uiAdsErrId			=> stMcAxisOnline.stHoldingBrake.uiAdsErrId,
					uiCANopenErrId		=> stMcAxisOnline.stHoldingBrake.uiSecErrId);
END_ACTION

